LIN {X 0,Y 467.586,Z 97.863,A -85,B 0,C 180,E1 -7602.569,E2 -7602.569} C_VEL
LIN {X 0,Y 467.57,Z 97.863,A -85,B 0,C 180,E1 -7605.055,E2 -7605.055} C_VEL
LIN {X 0,Y 467.589,Z 97.863,A -85,B 0,C 180,E1 -7607.442,E2 -7607.442} C_VEL
LIN {X 0,Y 467.56,Z 97.864,A -85,B 0,C 180,E1 -7610.855,E2 -7610.855} C_VEL
LIN {X 0,Y 467.56,Z 97.866,A -85,B 0,C 180,E1 -7614.263,E2 -7614.263} C_VEL
LIN {X 0,Y 467.582,Z 97.866,A -85,B 0,C 180,E1 -7617.323,E2 -7617.323} C_VEL
LIN {X 0,Y 467.57,Z 97.868,A -85,B 0,C 180,E1 -7620.67,E2 -7620.67} C_VEL
LIN {X 0,Y 467.644,Z 97.873,A -85,B 0,C 180,E1 -7622.313,E2 -7622.313} C_VEL
LIN {X 0,Y 470.573,Z 111.961,A -85,B 0,C 180,E1 -7624.81,E2 -7624.81} C_VEL
LIN {X 0,Y 470.522,Z 117.185,A -85,B 0,C 180,E1 -7625.665,E2 -7625.665} C_VEL
LIN {X 0,Y 469.718,Z 134.843,A -85,B 0,C 180,E1 -7628.497,E2 -7628.497} C_VEL
LIN {X 0,Y 469.444,Z 141.034,A -85,B 0,C 180,E1 -7629.471,E2 -7629.471} C_VEL
LIN {X 0,Y 473.187,Z 162.958,A -85,B 0,C 180,E1 -7629.971,E2 -7629.971} C_VEL
LIN {X 0,Y 471.968,Z 279.138,A -85,B 0,C 180,E1 -7631.779,E2 -7631.779} C_VEL
LIN {X 0,Y 471.559,Z 293.745,A -85,B 0,C 180,E1 -7632.184,E2 -7632.184} C_VEL
LIN {X 0,Y 471.065,Z 307.853,A -85,B 0,C 180,E1 -7632.759,E2 -7632.759} C_VEL
LIN {X 0,Y 470.402,Z 321.628,A -85,B 0,C 180,E1 -7633.51,E2 -7633.51} C_VEL
LIN {X 0,Y 469.751,Z 334.084,A -85,B 0,C 180,E1 -7634.379,E2 -7634.379} C_VEL
LIN {X 0,Y 469.073,Z 345.474,A -85,B 0,C 180,E1 -7635.356,E2 -7635.356} C_VEL
LIN {X 0,Y 468.461,Z 356.923,A -85,B 0,C 180,E1 -7636.555,E2 -7636.555} C_VEL
LIN {X 0,Y 467.959,Z 367.131,A -85,B 0,C 180,E1 -7637.864,E2 -7637.864} C_VEL
LIN {X 0,Y 467.506,Z 375.588,A -85,B 0,C 180,E1 -7639.17,E2 -7639.17} C_VEL
LIN {X 0,Y 467.122,Z 383.662,A -85,B 0,C 180,E1 -7640.694,E2 -7640.694} C_VEL
LIN {X 0,Y 466.853,Z 390.164,A -85,B 0,C 180,E1 -7642.215,E2 -7642.215} C_VEL
LIN {X 0,Y 466.709,Z 395.086,A -85,B 0,C 180,E1 -7643.66,E2 -7643.66} C_VEL
LIN {X 0,Y 466.721,Z 398.205,A -85,B 0,C 180,E1 -7644.818,E2 -7644.818} C_VEL
LIN {X 0,Y 466.652,Z 401.65,A -85,B 0,C 180,E1 -7646.548,E2 -7646.548} C_VEL
LIN {X 0,Y 466.607,Z 403.692,A -85,B 0,C 180,E1 -7648.275,E2 -7648.275} C_VEL
LIN {X 0,Y 466.601,Z 404.382,A -85,B 0,C 180,E1 -7650.001,E2 -7650.001} C_VEL
LIN {X 0,Y 466.607,Z 403.73,A -85,B 0,C 180,E1 -7651.727,E2 -7651.727} C_VEL
LIN {X 0,Y 466.653,Z 401.724,A -85,B 0,C 180,E1 -7653.455,E2 -7653.455} C_VEL
LIN {X 0,Y 466.722,Z 398.32,A -85,B 0,C 180,E1 -7655.185,E2 -7655.185} C_VEL
LIN {X 0,Y 466.827,Z 393.417,A -85,B 0,C 180,E1 -7656.919,E2 -7656.919} C_VEL
LIN {X 0,Y 467.025,Z 386.875,A -85,B 0,C 180,E1 -7658.656,E2 -7658.656} C_VEL
LIN {X 0,Y 467.304,Z 379.614,A -85,B 0,C 180,E1 -7660.18,E2 -7660.18} C_VEL
LIN {X 0,Y 467.839,Z 370.65,A -85,B 0,C 180,E1 -7661.702,E2 -7661.702} C_VEL
LIN {X 0,Y 468.33,Z 361.254,A -85,B 0,C 180,E1 -7663.01,E2 -7663.01} C_VEL
LIN {X 0,Y 468.911,Z 350.867,A -85,B 0,C 180,E1 -7664.208,E2 -7664.208} C_VEL
LIN {X 0,Y 469.603,Z 339.433,A -85,B 0,C 180,E1 -7665.295,E2 -7665.295} C_VEL
LIN {X 0,Y 470.358,Z 326.789,A -85,B 0,C 180,E1 -7666.271,E2 -7666.271} C_VEL
LIN {X 0,Y 471.062,Z 313.567,A -85,B 0,C 180,E1 -7667.08,E2 -7667.08} C_VEL
LIN {X 0,Y 471.608,Z 300.6,A -85,B 0,C 180,E1 -7667.694,E2 -7667.694} C_VEL
LIN {X 0,Y 472.129,Z 287.209,A -85,B 0,C 180,E1 -7668.155,E2 -7668.155} C_VEL
LIN {X 0,Y 472.522,Z 272.513,A -85,B 0,C 180,E1 -7668.482,E2 -7668.482} C_VEL
LIN {X 0,Y 473.546,Z 161.959,A -85,B 0,C 180,E1 -7670.211,E2 -7670.211} C_VEL
LIN {X 0,Y 469.646,Z 140.816,A -85,B 0,C 180,E1 -7670.746,E2 -7670.746} C_VEL
LIN {X 0,Y 470.621,Z 122.114,A -85,B 0,C 180,E1 -7673.78,E2 -7673.78} C_VEL
LIN {X 0,Y 471.062,Z 113.762,A -85,B 0,C 180,E1 -7675.165,E2 -7675.165} C_VEL
LIN {X 0,Y 468.091,Z 99.917,A -85,B 0,C 180,E1 -7677.74,E2 -7677.74} C_VEL
LIN {X 0,Y 467.62,Z 97.864,A -85,B 0,C 180,E1 -7678.136,E2 -7678.136} C_VEL
LIN {X 0,Y 467.593,Z 97.869,A -85,B 0,C 180,E1 -7681.741,E2 -7681.741} C_VEL
LIN {X 0,Y 467.568,Z 97.868,A -85,B 0,C 180,E1 -7684.834,E2 -7684.834} C_VEL
LIN {X 0,Y 467.574,Z 97.866,A -85,B 0,C 180,E1 -7688.045,E2 -7688.045} C_VEL
LIN {X 0,Y 467.586,Z 97.861,A -85,B 0,C 180,E1 -7691.403,E2 -7691.403} C_VEL
LIN {X 0,Y 467.579,Z 97.864,A -85,B 0,C 180,E1 -7695.052,E2 -7695.052} C_VEL
LIN {X 0,Y 467.588,Z 97.866,A -85,B 0,C 180,E1 -7697.438,E2 -7697.438} C_VEL
LIN {X 0,Y 467.582,Z 97.866,A -85,B 0,C 180,E1 -7700.047,E2 -7700.047} C_VEL
LIN {X 0,Y 467.537,Z 97.868,A -85,B 0,C 180,E1 -7703.036,E2 -7703.036} C_VEL
LIN {X 0,Y 467.582,Z 97.862,A -85,B 0,C 180,E1 -7706.209,E2 -7706.209} C_VEL
LIN {X 0,Y 467.581,Z 97.865,A -85,B 0,C 180,E1 -7709.265,E2 -7709.265} C_VEL
LIN {X 0,Y 467.617,Z 97.855,A -85,B 0,C 180,E1 -7712.468,E2 -7712.468} C_VEL
LIN {X 0,Y 467.596,Z 97.864,A -85,B 0,C 180,E1 -7715.11,E2 -7715.11} C_VEL
LIN {X 0,Y 467.547,Z 97.867,A -85,B 0,C 180,E1 -7717.925,E2 -7717.925} C_VEL
LIN {X 0,Y 467.634,Z 97.856,A -85,B 0,C 180,E1 -7720.69,E2 -7720.69} C_VEL
LIN {X 0,Y 467.65,Z 97.852,A -85,B 0,C 180,E1 -7724.303,E2 -7724.303} C_VEL
LIN {X 0,Y 467.668,Z 97.85,A -85,B 0,C 180,E1 -7727.852,E2 -7727.852} C_VEL
LIN {X 0,Y 467.677,Z 97.85,A -85,B 0,C 180,E1 -7731.355,E2 -7731.355} C_VEL
LIN {X 0,Y 467.721,Z 97.846,A -85,B 0,C 180,E1 -7733.96,E2 -7733.96} C_VEL
LIN {X 0,Y 467.858,Z 97.824,A -85,B 0,C 180,E1 -7737.414,E2 -7737.414} C_VEL
LIN {X 0,Y 467.887,Z 97.83,A -85,B 0,C 180,E1 -7739.997,E2 -7739.997} C_VEL
LIN {X 0,Y 467.857,Z 97.83,A -85,B 0,C 180,E1 -7742.58,E2 -7742.58} C_VEL
LIN {X 0,Y 467.725,Z 97.848,A -85,B 0,C 180,E1 -7746.035,E2 -7746.035} C_VEL
LIN {X 0,Y 467.672,Z 97.849,A -85,B 0,C 180,E1 -7748.64,E2 -7748.64} C_VEL
LIN {X 0,Y 467.658,Z 97.854,A -85,B 0,C 180,E1 -7752.142,E2 -7752.142} C_VEL
LIN {X 0,Y 467.638,Z 97.859,A -85,B 0,C 180,E1 -7755.692,E2 -7755.692} C_VEL
LIN {X 0,Y 467.619,Z 97.863,A -85,B 0,C 180,E1 -7759.304,E2 -7759.304} C_VEL
LIN {X 0,Y 467.53,Z 97.87,A -85,B 0,C 180,E1 -7762.07,E2 -7762.07} C_VEL
LIN {X 0,Y 467.563,Z 97.869,A -85,B 0,C 180,E1 -7764.886,E2 -7764.886} C_VEL
LIN {X 0,Y 467.608,Z 97.86,A -85,B 0,C 180,E1 -7767.766,E2 -7767.766} C_VEL
LIN {X 0,Y 467.557,Z 97.867,A -85,B 0,C 180,E1 -7771.041,E2 -7771.041} C_VEL
LIN {X 0,Y 467.565,Z 97.861,A -85,B 0,C 180,E1 -7774.236,E2 -7774.236} C_VEL
LIN {X 0,Y 467.532,Z 97.867,A -85,B 0,C 180,E1 -7777.182,E2 -7777.182} C_VEL
LIN {X 0,Y 467.558,Z 97.871,A -85,B 0,C 180,E1 -7780.261,E2 -7780.261} C_VEL
LIN {X 0,Y 467.569,Z 97.87,A -85,B 0,C 180,E1 -7782.563,E2 -7782.563} C_VEL
LIN {X 0,Y 467.546,Z 97.869,A -85,B 0,C 180,E1 -7785.049,E2 -7785.049} C_VEL
LIN {X 0,Y 467.551,Z 97.876,A -85,B 0,C 180,E1 -7788.593,E2 -7788.593} C_VEL
LIN {X 0,Y 467.605,Z 97.972,A -85,B 0,C 180,E1 -7789.323,E2 -7789.323} C_VEL
LIN {X 0,Y 469.891,Z 108.948,A -85,B 0,C 180,E1 -7791.631,E2 -7791.631} C_VEL
LIN {X 0,Y 470.21,Z 112.722,A -85,B 0,C 180,E1 -7792.381,E2 -7792.381} C_VEL
LIN {X 0,Y 469.959,Z 117.614,A -85,B 0,C 180,E1 -7793.306,E2 -7793.306} C_VEL
LIN {X 0,Y 473.812,Z 134.774,A -85,B 0,C 180,E1 -7793.792,E2 -7793.792} C_VEL
LIN {X 0,Y 472.582,Z 254.497,A -85,B 0,C 180,E1 -7795.685,E2 -7795.685} C_VEL
LIN {X 0,Y 472.2,Z 268.433,A -85,B 0,C 180,E1 -7796.073,E2 -7796.073} C_VEL
LIN {X 0,Y 472.044,Z 273.44,A -85,B 0,C 180,E1 -7796.253,E2 -7796.253} C_VEL
LIN {X 0,Y 471.249,Z 279.065,A -85,B 0,C 180,E1 -7796.453,E2 -7796.453} C_VEL
LIN {X 0,Y 468.134,Z 288.113,A -85,B 0,C 180,E1 -7796.775,E2 -7796.775} C_VEL
LIN {X 0,Y 464.937,Z 296.921,A -85,B 0,C 180,E1 -7797.179,E2 -7797.179} C_VEL
LIN {X 0,Y 464.02,Z 302.093,A -85,B 0,C 180,E1 -7797.502,E2 -7797.502} C_VEL
LIN {X 0,Y 463.276,Z 314.306,A -85,B 0,C 180,E1 -7798.461,E2 -7798.461} C_VEL
LIN {X 0,Y 462.579,Z 325.397,A -85,B 0,C 180,E1 -7799.53,E2 -7799.53} C_VEL
LIN {X 0,Y 461.928,Z 334.916,A -85,B 0,C 180,E1 -7800.631,E2 -7800.631} C_VEL
LIN {X 0,Y 461.223,Z 345.386,A -85,B 0,C 180,E1 -7802.093,E2 -7802.093} C_VEL
LIN {X 0,Y 460.703,Z 353.598,A -85,B 0,C 180,E1 -7803.498,E2 -7803.498} C_VEL
LIN {X 0,Y 460.305,Z 360.469,A -85,B 0,C 180,E1 -7804.931,E2 -7804.931} C_VEL
LIN {X 0,Y 459.964,Z 366.865,A -85,B 0,C 180,E1 -7806.591,E2 -7806.591} C_VEL
LIN {X 0,Y 459.825,Z 371.123,A -85,B 0,C 180,E1 -7808.008,E2 -7808.008} C_VEL
LIN {X 0,Y 459.653,Z 374.363,A -85,B 0,C 180,E1 -7809.41,E2 -7809.41} C_VEL
LIN {X 0,Y 459.492,Z 377.295,A -85,B 0,C 180,E1 -7811.263,E2 -7811.263} C_VEL
LIN {X 0,Y 459.422,Z 378.727,A -85,B 0,C 180,E1 -7813.102,E2 -7813.102} C_VEL
LIN {X 0,Y 459.471,Z 378.693,A -85,B 0,C 180,E1 -7814.927,E2 -7814.927} C_VEL
LIN {X 0,Y 459.477,Z 377.245,A -85,B 0,C 180,E1 -7816.735,E2 -7816.735} C_VEL
LIN {X 0,Y 459.622,Z 374.385,A -85,B 0,C 180,E1 -7818.533,E2 -7818.533} C_VEL
LIN {X 0,Y 459.756,Z 370.073,A -85,B 0,C 180,E1 -7820.319,E2 -7820.319} C_VEL
LIN {X 0,Y 460.008,Z 364.185,A -85,B 0,C 180,E1 -7822.095,E2 -7822.095} C_VEL
LIN {X 0,Y 460.358,Z 358.02,A -85,B 0,C 180,E1 -7823.544,E2 -7823.544} C_VEL
LIN {X 0,Y 460.723,Z 350.622,A -85,B 0,C 180,E1 -7824.967,E2 -7824.967} C_VEL
LIN {X 0,Y 461.238,Z 342.319,A -85,B 0,C 180,E1 -7826.286,E2 -7826.286} C_VEL
LIN {X 0,Y 461.841,Z 332.355,A -85,B 0,C 180,E1 -7827.6,E2 -7827.6} C_VEL
LIN {X 0,Y 462.503,Z 321.273,A -85,B 0,C 180,E1 -7828.802,E2 -7828.802} C_VEL
LIN {X 0,Y 463.207,Z 308.875,A -85,B 0,C 180,E1 -7829.89,E2 -7829.89} C_VEL
LIN {X 0,Y 463.947,Z 296.668,A -85,B 0,C 180,E1 -7830.752,E2 -7830.752} C_VEL
LIN {X 0,Y 464.499,Z 284.153,A -85,B 0,C 180,E1 -7831.456,E2 -7831.456} C_VEL
LIN {X 0,Y 464.951,Z 270.061,A -85,B 0,C 180,E1 -7832.056,E2 -7832.056} C_VEL
LIN {X 0,Y 465.269,Z 256.375,A -85,B 0,C 180,E1 -7832.461,E2 -7832.461} C_VEL
LIN {X 0,Y 465.598,Z 234.551,A -85,B 0,C 180,E1 -7832.838,E2 -7832.838} C_VEL
LIN {X 0,Y 466.531,Z 135.668,A -85,B 0,C 180,E1 -7834.384,E2 -7834.384} C_VEL
LIN {X 0,Y 462.773,Z 117.498,A -85,B 0,C 180,E1 -7834.858,E2 -7834.858} C_VEL
LIN {X 0,Y 462.996,Z 110.908,A -85,B 0,C 180,E1 -7836.098,E2 -7836.098} C_VEL
LIN {X 0,Y 460.643,Z 98.732,A -85,B 0,C 180,E1 -7838.592,E2 -7838.592} C_VEL
LIN {X 0,Y 460.633,Z 98.735,A -85,B 0,C 180,E1 -7842.478,E2 -7842.478} C_VEL
LIN {X 0,Y 460.583,Z 98.737,A -85,B 0,C 180,E1 -7846.007,E2 -7846.007} C_VEL
LIN {X 0,Y 460.538,Z 98.74,A -85,B 0,C 180,E1 -7848.904,E2 -7848.904} C_VEL
LIN {X 0,Y 460.527,Z 98.749,A -85,B 0,C 180,E1 -7851.484,E2 -7851.484} C_VEL
LIN {X 0,Y 460.522,Z 98.741,A -85,B 0,C 180,E1 -7854.332,E2 -7854.332} C_VEL
LIN {X 0,Y 460.548,Z 98.745,A -85,B 0,C 180,E1 -7857.244,E2 -7857.244} C_VEL
LIN {X 0,Y 460.498,Z 98.744,A -85,B 0,C 180,E1 -7860.239,E2 -7860.239} C_VEL
LIN {X 0,Y 460.495,Z 98.749,A -85,B 0,C 180,E1 -7863.326,E2 -7863.326} C_VEL
LIN {X 0,Y 460.475,Z 98.747,A -85,B 0,C 180,E1 -7866.018,E2 -7866.018} C_VEL
LIN {X 0,Y 460.559,Z 98.744,A -85,B 0,C 180,E1 -7868.907,E2 -7868.907} C_VEL
LIN {X 0,Y 460.517,Z 98.743,A -85,B 0,C 180,E1 -7872.18,E2 -7872.18} C_VEL
LIN {X 0,Y 460.525,Z 98.742,A -85,B 0,C 180,E1 -7875.418,E2 -7875.418} C_VEL
LIN {X 0,Y 460.516,Z 98.746,A -85,B 0,C 180,E1 -7878.397,E2 -7878.397} C_VEL
LIN {X 0,Y 460.523,Z 98.742,A -85,B 0,C 180,E1 -7881.272,E2 -7881.272} C_VEL
LIN {X 0,Y 460.487,Z 98.752,A -85,B 0,C 180,E1 -7884.557,E2 -7884.557} C_VEL
LIN {X 0,Y 460.507,Z 98.744,A -85,B 0,C 180,E1 -7887.718,E2 -7887.718} C_VEL
LIN {X 0,Y 460.523,Z 98.743,A -85,B 0,C 180,E1 -7890.772,E2 -7890.772} C_VEL
LIN {X 0,Y 460.561,Z 98.739,A -85,B 0,C 180,E1 -7893.739,E2 -7893.739} C_VEL
LIN {X 0,Y 460.539,Z 98.741,A -85,B 0,C 180,E1 -7896.628,E2 -7896.628} C_VEL
LIN {X 0,Y 460.553,Z 98.739,A -85,B 0,C 180,E1 -7899.457,E2 -7899.457} C_VEL
LIN {X 0,Y 460.541,Z 98.742,A -85,B 0,C 180,E1 -7902.233,E2 -7902.233} C_VEL
LIN {X 0,Y 460.552,Z 98.737,A -85,B 0,C 180,E1 -7904.968,E2 -7904.968} C_VEL
LIN {X 0,Y 460.613,Z 98.737,A -85,B 0,C 180,E1 -7907.669,E2 -7907.669} C_VEL
LIN {X 0,Y 460.616,Z 98.732,A -85,B 0,C 180,E1 -7911.227,E2 -7911.227} C_VEL
LIN {X 0,Y 460.701,Z 98.722,A -85,B 0,C 180,E1 -7913.873,E2 -7913.873} C_VEL
LIN {X 0,Y 460.815,Z 98.712,A -85,B 0,C 180,E1 -7917.381,E2 -7917.381} C_VEL
LIN {X 0,Y 460.842,Z 98.702,A -85,B 0,C 180,E1 -7920.003,E2 -7920.003} C_VEL
LIN {X 0,Y 460.816,Z 98.705,A -85,B 0,C 180,E1 -7922.625,E2 -7922.625} C_VEL
LIN {X 0,Y 460.701,Z 98.719,A -85,B 0,C 180,E1 -7926.133,E2 -7926.133} C_VEL
LIN {X 0,Y 460.621,Z 98.733,A -85,B 0,C 180,E1 -7928.779,E2 -7928.779} C_VEL
LIN {X 0,Y 460.606,Z 98.732,A -85,B 0,C 180,E1 -7932.448,E2 -7932.448} C_VEL
LIN {X 0,Y 460.594,Z 98.732,A -85,B 0,C 180,E1 -7936,E2 -7936} C_VEL
LIN {X 0,Y 460.566,Z 98.742,A -85,B 0,C 180,E1 -7938.904,E2 -7938.904} C_VEL
LIN {X 0,Y 460.511,Z 98.743,A -85,B 0,C 180,E1 -7941.488,E2 -7941.488} C_VEL
LIN {X 0,Y 460.539,Z 98.743,A -85,B 0,C 180,E1 -7944.335,E2 -7944.335} C_VEL
LIN {X 0,Y 460.581,Z 98.734,A -85,B 0,C 180,E1 -7947.245,E2 -7947.245} C_VEL
LIN {X 0,Y 460.508,Z 98.748,A -85,B 0,C 180,E1 -7950.242,E2 -7950.242} C_VEL
LIN {X 0,Y 460.527,Z 98.74,A -85,B 0,C 180,E1 -7953.327,E2 -7953.327} C_VEL
LIN {X 0,Y 460.476,Z 98.75,A -85,B 0,C 180,E1 -7956.532,E2 -7956.532} C_VEL
LIN {X 0,Y 460.531,Z 98.745,A -85,B 0,C 180,E1 -7959.865,E2 -7959.865} C_VEL
LIN {X 0,Y 460.512,Z 98.742,A -85,B 0,C 180,E1 -7962.902,E2 -7962.902} C_VEL
LIN {X 0,Y 460.509,Z 98.749,A -85,B 0,C 180,E1 -7965.833,E2 -7965.833} C_VEL
LIN {X 0,Y 460.531,Z 98.74,A -85,B 0,C 180,E1 -7968.991,E2 -7968.991} C_VEL
LIN {X 0,Y 460.519,Z 98.744,A -85,B 0,C 180,E1 -7971.268,E2 -7971.268} C_VEL
LIN {X 0,Y 460.511,Z 98.742,A -85,B 0,C 180,E1 -7974.556,E2 -7974.556} C_VEL
LIN {X 0,Y 460.532,Z 98.747,A -85,B 0,C 180,E1 -7977.717,E2 -7977.717} C_VEL
LIN {X 0,Y 460.54,Z 98.745,A -85,B 0,C 180,E1 -7980.771,E2 -7980.771} C_VEL
LIN {X 0,Y 460.602,Z 98.879,A -85,B 0,C 180,E1 -7982.094,E2 -7982.094} C_VEL
LIN {X 0,Y 463.594,Z 113.017,A -85,B 0,C 180,E1 -7984.644,E2 -7984.644} C_VEL
LIN {X 0,Y 463.751,Z 116.506,A -85,B 0,C 180,E1 -7985.234,E2 -7985.234} C_VEL
LIN {X 0,Y 462.737,Z 136.103,A -85,B 0,C 180,E1 -7988.424,E2 -7988.424} C_VEL
LIN {X 0,Y 462.521,Z 140.69,A -85,B 0,C 180,E1 -7989.164,E2 -7989.164} C_VEL
LIN {X 0,Y 466.435,Z 163.215,A -85,B 0,C 180,E1 -7989.702,E2 -7989.702} C_VEL
LIN {X 0,Y 465.217,Z 277.906,A -85,B 0,C 180,E1 -7991.505,E2 -7991.505} C_VEL
LIN {X 0,Y 464.833,Z 292.168,A -85,B 0,C 180,E1 -7991.888,E2 -7991.888} C_VEL
LIN {X 0,Y 464.265,Z 306.329,A -85,B 0,C 180,E1 -7992.455,E2 -7992.455} C_VEL
LIN {X 0,Y 463.639,Z 319.818,A -85,B 0,C 180,E1 -7993.182,E2 -7993.182} C_VEL
LIN {X 0,Y 462.962,Z 332.163,A -85,B 0,C 180,E1 -7994.031,E2 -7994.031} C_VEL
LIN {X 0,Y 462.252,Z 343.859,A -85,B 0,C 180,E1 -7995.022,E2 -7995.022} C_VEL
LIN {X 0,Y 461.592,Z 354.572,A -85,B 0,C 180,E1 -7996.126,E2 -7996.126} C_VEL
LIN {X 0,Y 461.074,Z 365.262,A -85,B 0,C 180,E1 -7997.465,E2 -7997.465} C_VEL
LIN {X 0,Y 460.553,Z 373.956,A -85,B 0,C 180,E1 -7998.782,E2 -7998.782} C_VEL
LIN {X 0,Y 460.116,Z 382.352,A -85,B 0,C 180,E1 -8000.329,E2 -8000.329} C_VEL
LIN {X 0,Y 459.846,Z 388.194,A -85,B 0,C 180,E1 -8001.653,E2 -8001.653} C_VEL
LIN {X 0,Y 459.735,Z 393.005,A -85,B 0,C 180,E1 -8002.977,E2 -8002.977} C_VEL
LIN {X 0,Y 459.628,Z 397.974,A -85,B 0,C 180,E1 -8004.737,E2 -8004.737} C_VEL
LIN {X 0,Y 459.55,Z 401.431,A -85,B 0,C 180,E1 -8006.494,E2 -8006.494} C_VEL
LIN {X 0,Y 459.52,Z 403.485,A -85,B 0,C 180,E1 -8008.248,E2 -8008.248} C_VEL
LIN {X 0,Y 459.533,Z 404.186,A -85,B 0,C 180,E1 -8010.001,E2 -8010.001} C_VEL
LIN {X 0,Y 459.52,Z 403.544,A -85,B 0,C 180,E1 -8011.754,E2 -8011.754} C_VEL
LIN {X 0,Y 459.549,Z 401.551,A -85,B 0,C 180,E1 -8013.508,E2 -8013.508} C_VEL
LIN {X 0,Y 459.63,Z 398.16,A -85,B 0,C 180,E1 -8015.265,E2 -8015.265} C_VEL
LIN {X 0,Y 459.738,Z 393.275,A -85,B 0,C 180,E1 -8017.026,E2 -8017.026} C_VEL
LIN {X 0,Y 459.96,Z 386.758,A -85,B 0,C 180,E1 -8018.79,E2 -8018.79} C_VEL
LIN {X 0,Y 460.275,Z 379.516,A -85,B 0,C 180,E1 -8020.337,E2 -8020.337} C_VEL
LIN {X 0,Y 460.832,Z 370.578,A -85,B 0,C 180,E1 -8021.882,E2 -8021.882} C_VEL
LIN {X 0,Y 461.349,Z 361.212,A -85,B 0,C 180,E1 -8023.21,E2 -8023.21} C_VEL
LIN {X 0,Y 462.004,Z 350.859,A -85,B 0,C 180,E1 -8024.425,E2 -8024.425} C_VEL
LIN {X 0,Y 462.719,Z 339.465,A -85,B 0,C 180,E1 -8025.528,E2 -8025.528} C_VEL
LIN {X 0,Y 463.549,Z 326.897,A -85,B 0,C 180,E1 -8026.517,E2 -8026.517} C_VEL
LIN {X 0,Y 464.269,Z 314.085,A -85,B 0,C 180,E1 -8027.321,E2 -8027.321} C_VEL
LIN {X 0,Y 464.928,Z 300.065,A -85,B 0,C 180,E1 -8027.997,E2 -8027.997} C_VEL
LIN {X 0,Y 465.476,Z 285.848,A -85,B 0,C 180,E1 -8028.487,E2 -8028.487} C_VEL
LIN {X 0,Y 465.878,Z 272.232,A -85,B 0,C 180,E1 -8028.784,E2 -8028.784} C_VEL
LIN {X 0,Y 467.066,Z 163.619,A -85,B 0,C 180,E1 -8030.502,E2 -8030.502} C_VEL
LIN {X 0,Y 463.42,Z 143.666,A -85,B 0,C 180,E1 -8031.017,E2 -8031.017} C_VEL
LIN {X 0,Y 462.796,Z 140.399,A -85,B 0,C 180,E1 -8031.119,E2 -8031.119} C_VEL
LIN {X 0,Y 463.853,Z 122.146,A -85,B 0,C 180,E1 -8034.149,E2 -8034.149} C_VEL
LIN {X 0,Y 464.183,Z 115.204,A -85,B 0,C 180,E1 -8035.324,E2 -8035.324} C_VEL
LIN {X 0,Y 461.509,Z 102.63,A -85,B 0,C 180,E1 -8037.702,E2 -8037.702} C_VEL
LIN {X 0,Y 460.584,Z 98.739,A -85,B 0,C 180,E1 -8038.48,E2 -8038.48} C_VEL
LIN {X 0,Y 460.532,Z 98.748,A -85,B 0,C 180,E1 -8041.283,E2 -8041.283} C_VEL
LIN {X 0,Y 460.534,Z 98.744,A -85,B 0,C 180,E1 -8044.504,E2 -8044.504} C_VEL
LIN {X 0,Y 460.511,Z 98.743,A -85,B 0,C 180,E1 -8047.624,E2 -8047.624} C_VEL
LIN {X 0,Y 460.54,Z 98.738,A -85,B 0,C 180,E1 -8051.012,E2 -8051.012} C_VEL
LIN {X 0,Y 460.525,Z 98.743,A -85,B 0,C 180,E1 -8054.589,E2 -8054.589} C_VEL
LIN {X 0,Y 460.527,Z 98.738,A -85,B 0,C 180,E1 -8057.817,E2 -8057.817} C_VEL
LIN {X 0,Y 460.531,Z 98.743,A -85,B 0,C 180,E1 -8060.135,E2 -8060.135} C_VEL
LIN {X 0,Y 460.486,Z 98.75,A -85,B 0,C 180,E1 -8063.469,E2 -8063.469} C_VEL
LIN {X 0,Y 460.532,Z 98.74,A -85,B 0,C 180,E1 -8066.673,E2 -8066.673} C_VEL
LIN {X 0,Y 460.52,Z 98.745,A -85,B 0,C 180,E1 -8069.759,E2 -8069.759} C_VEL
LIN {X 0,Y 460.548,Z 98.738,A -85,B 0,C 180,E1 -8072.752,E2 -8072.752} C_VEL
LIN {X 0,Y 460.542,Z 98.736,A -85,B 0,C 180,E1 -8075.665,E2 -8075.665} C_VEL
LIN {X 0,Y 460.535,Z 98.744,A -85,B 0,C 180,E1 -8078.577,E2 -8078.577} C_VEL
LIN {X 0,Y 460.597,Z 98.736,A -85,B 0,C 180,E1 -8081.309,E2 -8081.309} C_VEL
LIN {X 0,Y 460.617,Z 98.727,A -85,B 0,C 180,E1 -8084.057,E2 -8084.057} C_VEL
LIN {X 0,Y 460.621,Z 98.727,A -85,B 0,C 180,E1 -8087.664,E2 -8087.664} C_VEL
LIN {X 0,Y 460.628,Z 98.728,A -85,B 0,C 180,E1 -8091.221,E2 -8091.221} C_VEL
LIN {X 0,Y 460.686,Z 98.721,A -85,B 0,C 180,E1 -8093.867,E2 -8093.867} C_VEL
LIN {X 0,Y 460.799,Z 98.703,A -85,B 0,C 180,E1 -8097.375,E2 -8097.375} C_VEL
LIN {X 0,Y 460.857,Z 98.706,A -85,B 0,C 180,E1 -8099.997,E2 -8099.997} C_VEL
LIN {X 0,Y 460.797,Z 98.709,A -85,B 0,C 180,E1 -8102.62,E2 -8102.62} C_VEL
LIN {X 0,Y 460.689,Z 98.725,A -85,B 0,C 180,E1 -8106.127,E2 -8106.127} C_VEL
LIN {X 0,Y 460.623,Z 98.727,A -85,B 0,C 180,E1 -8108.773,E2 -8108.773} C_VEL
LIN {X 0,Y 460.611,Z 98.73,A -85,B 0,C 180,E1 -8112.331,E2 -8112.331} C_VEL
LIN {X 0,Y 460.6,Z 98.732,A -85,B 0,C 180,E1 -8115.994,E2 -8115.994} C_VEL
LIN {X 0,Y 460.565,Z 98.738,A -85,B 0,C 180,E1 -8119.612,E2 -8119.612} C_VEL
LIN {X 0,Y 460.506,Z 98.744,A -85,B 0,C 180,E1 -8122.425,E2 -8122.425} C_VEL
LIN {X 0,Y 460.539,Z 98.739,A -85,B 0,C 180,E1 -8125.792,E2 -8125.792} C_VEL
LIN {X 0,Y 460.541,Z 98.74,A -85,B 0,C 180,E1 -8128.229,E2 -8128.229} C_VEL
LIN {X 0,Y 460.51,Z 98.748,A -85,B 0,C 180,E1 -8131.279,E2 -8131.279} C_VEL
LIN {X 0,Y 460.51,Z 98.74,A -85,B 0,C 180,E1 -8134.5,E2 -8134.5} C_VEL
LIN {X 0,Y 460.486,Z 98.743,A -85,B 0,C 180,E1 -8137.619,E2 -8137.619} C_VEL
LIN {X 0,Y 460.522,Z 98.747,A -85,B 0,C 180,E1 -8140.265,E2 -8140.265} C_VEL
LIN {X 0,Y 460.48,Z 98.75,A -85,B 0,C 180,E1 -8143.372,E2 -8143.372} C_VEL
LIN {X 0,Y 460.488,Z 98.754,A -85,B 0,C 180,E1 -8146.622,E2 -8146.622} C_VEL
LIN {X 0,Y 460.555,Z 98.89,A -85,B 0,C 180,E1 -8149.024,E2 -8149.024} C_VEL
LIN {X 0,Y 463.004,Z 110.519,A -85,B 0,C 180,E1 -8151.511,E2 -8151.511} C_VEL
LIN {X 0,Y 463.325,Z 114.669,A -85,B 0,C 180,E1 -8152.348,E2 -8152.348} C_VEL
LIN {X 0,Y 463.133,Z 117.901,A -85,B 0,C 180,E1 -8152.967,E2 -8152.967} C_VEL
LIN {X 0,Y 467.31,Z 136.33,A -85,B 0,C 180,E1 -8153.49,E2 -8153.49} C_VEL
LIN {X 0,Y 465.932,Z 254.799,A -85,B 0,C 180,E1 -8155.388,E2 -8155.388} C_VEL
LIN {X 0,Y 465.545,Z 268.701,A -85,B 0,C 180,E1 -8155.781,E2 -8155.781} C_VEL
LIN {X 0,Y 465.038,Z 282.141,A -85,B 0,C 180,E1 -8156.333,E2 -8156.333} C_VEL
LIN {X 0,Y 464.336,Z 296.242,A -85,B 0,C 180,E1 -8157.111,E2 -8157.111} C_VEL
LIN {X 0,Y 464.02,Z 302.093,A -85,B 0,C 180,E1 -8157.502,E2 -8157.502} C_VEL
LIN {X 0,Y 463.111,Z 307.223,A -85,B 0,C 180,E1 -8157.852,E2 -8157.852} C_VEL
LIN {X 0,Y 459.89,Z 315.403,A -85,B 0,C 180,E1 -8158.417,E2 -8158.417} C_VEL
LIN {X 0,Y 456.59,Z 323.242,A -85,B 0,C 180,E1 -8159.055,E2 -8159.055} C_VEL
LIN {X 0,Y 455.571,Z 327.76,A -85,B 0,C 180,E1 -8159.513,E2 -8159.513} C_VEL
LIN {X 0,Y 454.929,Z 336.909,A -85,B 0,C 180,E1 -8160.626,E2 -8160.626} C_VEL
LIN {X 0,Y 454.193,Z 346.884,A -85,B 0,C 180,E1 -8162.093,E2 -8162.093} C_VEL
LIN {X 0,Y 453.587,Z 355.724,A -85,B 0,C 180,E1 -8163.697,E2 -8163.697} C_VEL
LIN {X 0,Y 453.139,Z 362.605,A -85,B 0,C 180,E1 -8165.243,E2 -8165.243} C_VEL
LIN {X 0,Y 452.89,Z 367.88,A -85,B 0,C 180,E1 -8166.713,E2 -8166.713} C_VEL
LIN {X 0,Y 452.736,Z 371.923,A -85,B 0,C 180,E1 -8168.125,E2 -8168.125} C_VEL
LIN {X 0,Y 452.607,Z 374.082,A -85,B 0,C 180,E1 -8169.074,E2 -8169.074} C_VEL
LIN {X 0,Y 452.402,Z 377.194,A -85,B 0,C 180,E1 -8170.959,E2 -8170.959} C_VEL
LIN {X 0,Y 452.327,Z 378.799,A -85,B 0,C 180,E1 -8172.829,E2 -8172.829} C_VEL
LIN {X 0,Y 452.383,Z 378.963,A -85,B 0,C 180,E1 -8174.685,E2 -8174.685} C_VEL
LIN {X 0,Y 452.376,Z 377.721,A -85,B 0,C 180,E1 -8176.523,E2 -8176.523} C_VEL
LIN {X 0,Y 452.528,Z 375.04,A -85,B 0,C 180,E1 -8178.351,E2 -8178.351} C_VEL
LIN {X 0,Y 452.655,Z 370.903,A -85,B 0,C 180,E1 -8180.165,E2 -8180.165} C_VEL
LIN {X 0,Y 452.907,Z 365.201,A -85,B 0,C 180,E1 -8181.971,E2 -8181.971} C_VEL
LIN {X 0,Y 453.278,Z 359.02,A -85,B 0,C 180,E1 -8183.49,E2 -8183.49} C_VEL
LIN {X 0,Y 453.699,Z 350.836,A -85,B 0,C 180,E1 -8185.111,E2 -8185.111} C_VEL
LIN {X 0,Y 454.267,Z 342.53,A -85,B 0,C 180,E1 -8186.451,E2 -8186.451} C_VEL
LIN {X 0,Y 454.893,Z 332.564,A -85,B 0,C 180,E1 -8187.785,E2 -8187.785} C_VEL
LIN {X 0,Y 455.586,Z 321.471,A -85,B 0,C 180,E1 -8189.004,E2 -8189.004} C_VEL
LIN {X 0,Y 456.332,Z 308.914,A -85,B 0,C 180,E1 -8190.12,E2 -8190.12} C_VEL
LIN {X 0,Y 457.12,Z 295.753,A -85,B 0,C 180,E1 -8191.052,E2 -8191.052} C_VEL
LIN {X 0,Y 457.736,Z 283.043,A -85,B 0,C 180,E1 -8191.758,E2 -8191.758} C_VEL
LIN {X 0,Y 458.179,Z 268.659,A -85,B 0,C 180,E1 -8192.361,E2 -8192.361} C_VEL
LIN {X 0,Y 458.549,Z 254.092,A -85,B 0,C 180,E1 -8192.771,E2 -8192.771} C_VEL
LIN {X 0,Y 459.848,Z 136.88,A -85,B 0,C 180,E1 -8194.647,E2 -8194.647} C_VEL
LIN {X 0,Y 455.871,Z 117.738,A -85,B 0,C 180,E1 -8195.144,E2 -8195.144} C_VEL
LIN {X 0,Y 456.072,Z 112.259,A -85,B 0,C 180,E1 -8196.191,E2 -8196.191} C_VEL
LIN {X 0,Y 453.582,Z 99.611,A -85,B 0,C 180,E1 -8198.82,E2 -8198.82} C_VEL
LIN {X 0,Y 453.602,Z 99.611,A -85,B 0,C 180,E1 -8202.572,E2 -8202.572} C_VEL
LIN {X 0,Y 453.52,Z 99.615,A -85,B 0,C 180,E1 -8206.195,E2 -8206.195} C_VEL
LIN {X 0,Y 453.487,Z 99.619,A -85,B 0,C 180,E1 -8209.043,E2 -8209.043} C_VEL
LIN {X 0,Y 453.468,Z 99.623,A -85,B 0,C 180,E1 -8211.835,E2 -8211.835} C_VEL
LIN {X 0,Y 453.496,Z 99.617,A -85,B 0,C 180,E1 -8214.734,E2 -8214.734} C_VEL
LIN {X 0,Y 453.502,Z 99.616,A -85,B 0,C 180,E1 -8217.962,E2 -8217.962} C_VEL
LIN {X 0,Y 453.45,Z 99.625,A -85,B 0,C 180,E1 -8220.76,E2 -8220.76} C_VEL
LIN {X 0,Y 453.446,Z 99.623,A -85,B 0,C 180,E1 -8223.914,E2 -8223.914} C_VEL
LIN {X 0,Y 453.447,Z 99.628,A -85,B 0,C 180,E1 -8227.188,E2 -8227.188} C_VEL
LIN {X 0,Y 453.511,Z 99.616,A -85,B 0,C 180,E1 -8229.446,E2 -8229.446} C_VEL
LIN {X 0,Y 453.468,Z 99.625,A -85,B 0,C 180,E1 -8232.992,E2 -8232.992} C_VEL
LIN {X 0,Y 453.511,Z 99.614,A -85,B 0,C 180,E1 -8235.791,E2 -8235.791} C_VEL
LIN {X 0,Y 453.487,Z 99.618,A -85,B 0,C 180,E1 -8239.408,E2 -8239.408} C_VEL
LIN {X 0,Y 453.451,Z 99.626,A -85,B 0,C 180,E1 -8242.224,E2 -8242.224} C_VEL
LIN {X 0,Y 453.462,Z 99.621,A -85,B 0,C 180,E1 -8245.225,E2 -8245.225} C_VEL
LIN {X 0,Y 453.459,Z 99.627,A -85,B 0,C 180,E1 -8248.473,E2 -8248.473} C_VEL
LIN {X 0,Y 453.491,Z 99.617,A -85,B 0,C 180,E1 -8251.291,E2 -8251.291} C_VEL
LIN {X 0,Y 453.532,Z 99.618,A -85,B 0,C 180,E1 -8254.289,E2 -8254.289} C_VEL
LIN {X 0,Y 453.48,Z 99.618,A -85,B 0,C 180,E1 -8257.208,E2 -8257.208} C_VEL
LIN {X 0,Y 453.508,Z 99.621,A -85,B 0,C 180,E1 -8260.07,E2 -8260.07} C_VEL
LIN {X 0,Y 453.491,Z 99.617,A -85,B 0,C 180,E1 -8262.879,E2 -8262.879} C_VEL
LIN {X 0,Y 453.498,Z 99.622,A -85,B 0,C 180,E1 -8265.647,E2 -8265.647} C_VEL
LIN {X 0,Y 453.564,Z 99.609,A -85,B 0,C 180,E1 -8268.382,E2 -8268.382} C_VEL
LIN {X 0,Y 453.637,Z 99.602,A -85,B 0,C 180,E1 -8271.988,E2 -8271.988} C_VEL
LIN {X 0,Y 453.663,Z 99.596,A -85,B 0,C 180,E1 -8274.67,E2 -8274.67} C_VEL
LIN {X 0,Y 453.756,Z 99.591,A -85,B 0,C 180,E1 -8277.34,E2 -8277.34} C_VEL
LIN {X 0,Y 453.813,Z 99.578,A -85,B 0,C 180,E1 -8280.003,E2 -8280.003} C_VEL
LIN {X 0,Y 453.756,Z 99.585,A -85,B 0,C 180,E1 -8282.666,E2 -8282.666} C_VEL
LIN {X 0,Y 453.669,Z 99.595,A -85,B 0,C 180,E1 -8286.228,E2 -8286.228} C_VEL
LIN {X 0,Y 453.584,Z 99.611,A -85,B 0,C 180,E1 -8288.916,E2 -8288.916} C_VEL
LIN {X 0,Y 453.556,Z 99.611,A -85,B 0,C 180,E1 -8292.532,E2 -8292.532} C_VEL
LIN {X 0,Y 453.539,Z 99.612,A -85,B 0,C 180,E1 -8296.199,E2 -8296.199} C_VEL
LIN {X 0,Y 453.515,Z 99.618,A -85,B 0,C 180,E1 -8299.043,E2 -8299.043} C_VEL
LIN {X 0,Y 453.472,Z 99.619,A -85,B 0,C 180,E1 -8301.839,E2 -8301.839} C_VEL
LIN {X 0,Y 453.511,Z 99.62,A -85,B 0,C 180,E1 -8304.737,E2 -8304.737} C_VEL
LIN {X 0,Y 453.534,Z 99.613,A -85,B 0,C 180,E1 -8307.963,E2 -8307.963} C_VEL
LIN {X 0,Y 453.463,Z 99.621,A -85,B 0,C 180,E1 -8311.527,E2 -8311.527} C_VEL
LIN {X 0,Y 453.487,Z 99.619,A -85,B 0,C 180,E1 -8314.78,E2 -8314.78} C_VEL
LIN {X 0,Y 453.463,Z 99.626,A -85,B 0,C 180,E1 -8318.314,E2 -8318.314} C_VEL
LIN {X 0,Y 453.493,Z 99.618,A -85,B 0,C 180,E1 -8320.611,E2 -8320.611} C_VEL
LIN {X 0,Y 453.455,Z 99.622,A -85,B 0,C 180,E1 -8323.246,E2 -8323.246} C_VEL
LIN {X 0,Y 453.464,Z 99.626,A -85,B 0,C 180,E1 -8325.781,E2 -8325.781} C_VEL
LIN {X 0,Y 453.479,Z 99.622,A -85,B 0,C 180,E1 -8328.211,E2 -8328.211} C_VEL
LIN {X 0,Y 453.472,Z 99.619,A -85,B 0,C 180,E1 -8330.799,E2 -8330.799} C_VEL
LIN {X 0,Y 453.455,Z 99.626,A -85,B 0,C 180,E1 -8333.919,E2 -8333.919} C_VEL
LIN {X 0,Y 453.483,Z 99.621,A -85,B 0,C 180,E1 -8337.153,E2 -8337.153} C_VEL
LIN {X 0,Y 453.475,Z 99.624,A -85,B 0,C 180,E1 -8340.27,E2 -8340.27} C_VEL
LIN {X 0,Y 453.538,Z 99.695,A -85,B 0,C 180,E1 -8341.84,E2 -8341.84} C_VEL
LIN {X 0,Y 456.58,Z 114.037,A -85,B 0,C 180,E1 -8344.471,E2 -8344.471} C_VEL
LIN {X 0,Y 456.927,Z 116.578,A -85,B 0,C 180,E1 -8344.918,E2 -8344.918} C_VEL
LIN {X 0,Y 455.777,Z 136.95,A -85,B 0,C 180,E1 -8348.281,E2 -8348.281} C_VEL
LIN {X 0,Y 455.6,Z 140.516,A -85,B 0,C 180,E1 -8348.866,E2 -8348.866} C_VEL
LIN {X 0,Y 459.708,Z 164.556,A -85,B 0,C 180,E1 -8349.445,E2 -8349.445} C_VEL
LIN {X 0,Y 458.396,Z 278.976,A -85,B 0,C 180,E1 -8351.278,E2 -8351.278} C_VEL
LIN {X 0,Y 457.952,Z 293.523,A -85,B 0,C 180,E1 -8351.693,E2 -8351.693} C_VEL
LIN {X 0,Y 457.385,Z 307.133,A -85,B 0,C 180,E1 -8352.26,E2 -8352.26} C_VEL
LIN {X 0,Y 456.739,Z 320.478,A -85,B 0,C 180,E1 -8353.002,E2 -8353.002} C_VEL
LIN {X 0,Y 455.977,Z 333.093,A -85,B 0,C 180,E1 -8353.894,E2 -8353.894} C_VEL
LIN {X 0,Y 455.171,Z 345.788,A -85,B 0,C 180,E1 -8355.013,E2 -8355.013} C_VEL
LIN {X 0,Y 454.517,Z 356.145,A -85,B 0,C 180,E1 -8356.134,E2 -8356.134} C_VEL
LIN {X 0,Y 453.976,Z 366.439,A -85,B 0,C 180,E1 -8357.484,E2 -8357.484} C_VEL
LIN {X 0,Y 453.445,Z 374.956,A -85,B 0,C 180,E1 -8358.83,E2 -8358.83} C_VEL
LIN {X 0,Y 453.032,Z 383.084,A -85,B 0,C 180,E1 -8360.401,E2 -8360.401} C_VEL
LIN {X 0,Y 452.721,Z 389.629,A -85,B 0,C 180,E1 -8361.97,E2 -8361.97} C_VEL
LIN {X 0,Y 452.583,Z 394.17,A -85,B 0,C 180,E1 -8363.314,E2 -8363.314} C_VEL
LIN {X 0,Y 452.537,Z 397.726,A -85,B 0,C 180,E1 -8364.655,E2 -8364.655} C_VEL
LIN {X 0,Y 452.448,Z 401.2,A -85,B 0,C 180,E1 -8366.439,E2 -8366.439} C_VEL
LIN {X 0,Y 452.502,Z 402.409,A -85,B 0,C 180,E1 -8367.331,E2 -8367.331} C_VEL
LIN {X 0,Y 452.428,Z 403.796,A -85,B 0,C 180,E1 -8369.111,E2 -8369.111} C_VEL
LIN {X 0,Y 452.428,Z 403.842,A -85,B 0,C 180,E1 -8370.891,E2 -8370.891} C_VEL
LIN {X 0,Y 452.503,Z 402.548,A -85,B 0,C 180,E1 -8372.672,E2 -8372.672} C_VEL
LIN {X 0,Y 452.471,Z 399.879,A -85,B 0,C 180,E1 -8374.455,E2 -8374.455} C_VEL
LIN {X 0,Y 452.57,Z 395.771,A -85,B 0,C 180,E1 -8376.242,E2 -8376.242} C_VEL
LIN {X 0,Y 452.744,Z 390.106,A -85,B 0,C 180,E1 -8378.032,E2 -8378.032} C_VEL
LIN {X 0,Y 453.055,Z 383.729,A -85,B 0,C 180,E1 -8379.601,E2 -8379.601} C_VEL
LIN {X 0,Y 453.514,Z 375.81,A -85,B 0,C 180,E1 -8381.171,E2 -8381.171} C_VEL
LIN {X 0,Y 454.048,Z 366.797,A -85,B 0,C 180,E1 -8382.633,E2 -8382.633} C_VEL
LIN {X 0,Y 454.636,Z 357.639,A -85,B 0,C 180,E1 -8383.865,E2 -8383.865} C_VEL
LIN {X 0,Y 455.386,Z 346.632,A -85,B 0,C 180,E1 -8385.097,E2 -8385.097} C_VEL
LIN {X 0,Y 456.297,Z 334.387,A -85,B 0,C 180,E1 -8386.212,E2 -8386.212} C_VEL
LIN {X 0,Y 457.089,Z 321.518,A -85,B 0,C 180,E1 -8387.152,E2 -8387.152} C_VEL
LIN {X 0,Y 457.872,Z 307.747,A -85,B 0,C 180,E1 -8387.937,E2 -8387.937} C_VEL
LIN {X 0,Y 458.49,Z 293.396,A -85,B 0,C 180,E1 -8388.547,E2 -8388.547} C_VEL
LIN {X 0,Y 459.039,Z 279.106,A -85,B 0,C 180,E1 -8388.959,E2 -8388.959} C_VEL
LIN {X 0,Y 459.859,Z 218.509,A -85,B 0,C 180,E1 -8389.953,E2 -8389.953} C_VEL
LIN {X 0,Y 460.4,Z 163.646,A -85,B 0,C 180,E1 -8390.84,E2 -8390.84} C_VEL
LIN {X 0,Y 456.742,Z 144.122,A -85,B 0,C 180,E1 -8391.364,E2 -8391.364} C_VEL
LIN {X 0,Y 455.964,Z 140.166,A -85,B 0,C 180,E1 -8391.492,E2 -8391.492} C_VEL
LIN {X 0,Y 457.111,Z 122.198,A -85,B 0,C 180,E1 -8394.528,E2 -8394.528} C_VEL
LIN {X 0,Y 457.308,Z 116.642,A -85,B 0,C 180,E1 -8395.488,E2 -8395.488} C_VEL
LIN {X 0,Y 454.965,Z 105.629,A -85,B 0,C 180,E1 -8397.609,E2 -8397.609} C_VEL
LIN {X 0,Y 453.518,Z 99.618,A -85,B 0,C 180,E1 -8398.839,E2 -8398.839} C_VEL
LIN {X 0,Y 453.475,Z 99.628,A -85,B 0,C 180,E1 -8401.8,E2 -8401.8} C_VEL
LIN {X 0,Y 453.488,Z 99.622,A -85,B 0,C 180,E1 -8404.99,E2 -8404.99} C_VEL
LIN {X 0,Y 453.47,Z 99.626,A -85,B 0,C 180,E1 -8408.312,E2 -8408.312} C_VEL
LIN {X 0,Y 453.507,Z 99.614,A -85,B 0,C 180,E1 -8410.609,E2 -8410.609} C_VEL
LIN {X 0,Y 453.473,Z 99.625,A -85,B 0,C 180,E1 -8414.222,E2 -8414.222} C_VEL
LIN {X 0,Y 453.475,Z 99.622,A -85,B 0,C 180,E1 -8417.004,E2 -8417.004} C_VEL
LIN {X 0,Y 453.507,Z 99.608,A -85,B 0,C 180,E1 -8419.409,E2 -8419.409} C_VEL
LIN {X 0,Y 453.463,Z 99.62,A -85,B 0,C 180,E1 -8422.809,E2 -8422.809} C_VEL
LIN {X 0,Y 453.481,Z 99.619,A -85,B 0,C 180,E1 -8426.086,E2 -8426.086} C_VEL
LIN {X 0,Y 453.489,Z 99.62,A -85,B 0,C 180,E1 -8429.239,E2 -8429.239} C_VEL
LIN {X 0,Y 453.521,Z 99.611,A -85,B 0,C 180,E1 -8432.294,E2 -8432.294} C_VEL
LIN {X 0,Y 453.513,Z 99.616,A -85,B 0,C 180,E1 -8435.263,E2 -8435.263} C_VEL
LIN {X 0,Y 453.494,Z 99.619,A -85,B 0,C 180,E1 -8438.413,E2 -8438.413} C_VEL
LIN {X 0,Y 453.535,Z 99.617,A -85,B 0,C 180,E1 -8441.007,E2 -8441.007} C_VEL
LIN {X 0,Y 453.582,Z 99.602,A -85,B 0,C 180,E1 -8443.878,E2 -8443.878} C_VEL
LIN {X 0,Y 453.576,Z 99.605,A -85,B 0,C 180,E1 -8447.469,E2 -8447.469} C_VEL
LIN {X 0,Y 453.594,Z 99.605,A -85,B 0,C 180,E1 -8451.084,E2 -8451.084} C_VEL
LIN {X 0,Y 453.652,Z 99.597,A -85,B 0,C 180,E1 -8453.772,E2 -8453.772} C_VEL
LIN {X 0,Y 453.743,Z 99.582,A -85,B 0,C 180,E1 -8457.334,E2 -8457.334} C_VEL
LIN {X 0,Y 453.827,Z 99.581,A -85,B 0,C 180,E1 -8459.997,E2 -8459.997} C_VEL
LIN {X 0,Y 453.741,Z 99.588,A -85,B 0,C 180,E1 -8462.66,E2 -8462.66} C_VEL
LIN {X 0,Y 453.655,Z 99.601,A -85,B 0,C 180,E1 -8466.222,E2 -8466.222} C_VEL
LIN {X 0,Y 453.588,Z 99.604,A -85,B 0,C 180,E1 -8468.91,E2 -8468.91} C_VEL
LIN {X 0,Y 453.566,Z 99.607,A -85,B 0,C 180,E1 -8472.525,E2 -8472.525} C_VEL
LIN {X 0,Y 453.544,Z 99.609,A -85,B 0,C 180,E1 -8476.192,E2 -8476.192} C_VEL
LIN {X 0,Y 453.514,Z 99.619,A -85,B 0,C 180,E1 -8479.035,E2 -8479.035} C_VEL
LIN {X 0,Y 453.473,Z 99.622,A -85,B 0,C 180,E1 -8481.832,E2 -8481.832} C_VEL
LIN {X 0,Y 453.486,Z 99.621,A -85,B 0,C 180,E1 -8484.732,E2 -8484.732} C_VEL
LIN {X 0,Y 453.521,Z 99.615,A -85,B 0,C 180,E1 -8487.955,E2 -8487.955} C_VEL
LIN {X 0,Y 453.454,Z 99.625,A -85,B 0,C 180,E1 -8491.521,E2 -8491.521} C_VEL
LIN {X 0,Y 453.47,Z 99.619,A -85,B 0,C 180,E1 -8494.772,E2 -8494.772} C_VEL
LIN {X 0,Y 453.447,Z 99.622,A -85,B 0,C 180,E1 -8498.308,E2 -8498.308} C_VEL
LIN {X 0,Y 453.478,Z 99.621,A -85,B 0,C 180,E1 -8500.605,E2 -8500.605} C_VEL
LIN {X 0,Y 453.437,Z 99.628,A -85,B 0,C 180,E1 -8503.24,E2 -8503.24} C_VEL
LIN {X 0,Y 453.44,Z 99.626,A -85,B 0,C 180,E1 -8505.774,E2 -8505.774} C_VEL
LIN {X 0,Y 453.518,Z 99.798,A -85,B 0,C 180,E1 -8508.706,E2 -8508.706} C_VEL
LIN {X 0,Y 456.061,Z 111.805,A -85,B 0,C 180,E1 -8511.329,E2 -8511.329} C_VEL
LIN {X 0,Y 456.514,Z 114.962,A -85,B 0,C 180,E1 -8511.989,E2 -8511.989} C_VEL
LIN {X 0,Y 456.389,Z 118.299,A -85,B 0,C 180,E1 -8512.606,E2 -8512.606} C_VEL
LIN {X 0,Y 460.753,Z 137.386,A -85,B 0,C 180,E1 -8513.166,E2 -8513.166} C_VEL
LIN {X 0,Y 459.299,Z 255.112,A -85,B 0,C 180,E1 -8515.083,E2 -8515.083} C_VEL
LIN {X 0,Y 458.86,Z 269.379,A -85,B 0,C 180,E1 -8515.495,E2 -8515.495} C_VEL
LIN {X 0,Y 458.342,Z 282.597,A -85,B 0,C 180,E1 -8516.05,E2 -8516.05} C_VEL
LIN {X 0,Y 457.614,Z 296.474,A -85,B 0,C 180,E1 -8516.829,E2 -8516.829} C_VEL
LIN {X 0,Y 456.819,Z 309.72,A -85,B 0,C 180,E1 -8517.787,E2 -8517.787} C_VEL
LIN {X 0,Y 455.985,Z 322.125,A -85,B 0,C 180,E1 -8518.912,E2 -8518.912} C_VEL
LIN {X 0,Y 455.571,Z 327.76,A -85,B 0,C 180,E1 -8519.513,E2 -8519.513} C_VEL
LIN {X 0,Y 454.55,Z 332.181,A -85,B 0,C 180,E1 -8519.998,E2 -8519.998} C_VEL
LIN {X 0,Y 451.222,Z 339.102,A -85,B 0,C 180,E1 -8520.794,E2 -8520.794} C_VEL
LIN {X 0,Y 447.975,Z 345.598,A -85,B 0,C 180,E1 -8521.655,E2 -8521.655} C_VEL
LIN {X 0,Y 447.084,Z 349.201,A -85,B 0,C 180,E1 -8522.235,E2 -8522.235} C_VEL
LIN {X 0,Y 446.483,Z 357.588,A -85,B 0,C 180,E1 -8523.847,E2 -8523.847} C_VEL
LIN {X 0,Y 446.056,Z 363.772,A -85,B 0,C 180,E1 -8525.32,E2 -8525.32} C_VEL
LIN {X 0,Y 445.819,Z 368.757,A -85,B 0,C 180,E1 -8526.789,E2 -8526.789} C_VEL
LIN {X 0,Y 445.605,Z 373.282,A -85,B 0,C 180,E1 -8528.505,E2 -8528.505} C_VEL
LIN {X 0,Y 445.42,Z 375.647,A -85,B 0,C 180,E1 -8529.687,E2 -8529.687} C_VEL
LIN {X 0,Y 445.31,Z 378.167,A -85,B 0,C 180,E1 -8531.599,E2 -8531.599} C_VEL
LIN {X 0,Y 445.239,Z 379.215,A -85,B 0,C 180,E1 -8533.492,E2 -8533.492} C_VEL
LIN {X 0,Y 445.271,Z 378.839,A -85,B 0,C 180,E1 -8535.371,E2 -8535.371} C_VEL
LIN {X 0,Y 445.323,Z 377.066,A -85,B 0,C 180,E1 -8537.234,E2 -8537.234} C_VEL
LIN {X 0,Y 445.498,Z 373.877,A -85,B 0,C 180,E1 -8539.086,E2 -8539.086} C_VEL
LIN {X 0,Y 445.661,Z 369.173,A -85,B 0,C 180,E1 -8540.925,E2 -8540.925} C_VEL
LIN {X 0,Y 445.907,Z 364.585,A -85,B 0,C 180,E1 -8542.3,E2 -8542.3} C_VEL
LIN {X 0,Y 446.237,Z 357.97,A -85,B 0,C 180,E1 -8543.896,E2 -8543.896} C_VEL
LIN {X 0,Y 446.729,Z 349.759,A -85,B 0,C 180,E1 -8545.487,E2 -8545.487} C_VEL
LIN {X 0,Y 447.356,Z 341.187,A -85,B 0,C 180,E1 -8546.847,E2 -8546.847} C_VEL
LIN {X 0,Y 448.067,Z 330.836,A -85,B 0,C 180,E1 -8548.201,E2 -8548.201} C_VEL
LIN {X 0,Y 448.754,Z 320.455,A -85,B 0,C 180,E1 -8549.326,E2 -8549.326} C_VEL
LIN {X 0,Y 449.455,Z 309.184,A -85,B 0,C 180,E1 -8550.335,E2 -8550.335} C_VEL
LIN {X 0,Y 450.28,Z 296.019,A -85,B 0,C 180,E1 -8551.282,E2 -8551.282} C_VEL
LIN {X 0,Y 450.909,Z 283.15,A -85,B 0,C 180,E1 -8552.008,E2 -8552.008} C_VEL
LIN {X 0,Y 451.348,Z 269.488,A -85,B 0,C 180,E1 -8552.592,E2 -8552.592} C_VEL
LIN {X 0,Y 451.692,Z 255.322,A -85,B 0,C 180,E1 -8553.009,E2 -8553.009} C_VEL
LIN {X 0,Y 452.838,Z 164.005,A -85,B 0,C 180,E1 -8554.5,E2 -8554.5} C_VEL
LIN {X 0,Y 453.072,Z 137.708,A -85,B 0,C 180,E1 -8554.926,E2 -8554.926} C_VEL
LIN {X 0,Y 448.941,Z 117.946,A -85,B 0,C 180,E1 -8555.445,E2 -8555.445} C_VEL
LIN {X 0,Y 449.138,Z 113.586,A -85,B 0,C 180,E1 -8556.287,E2 -8556.287} C_VEL
LIN {X 0,Y 446.555,Z 100.486,A -85,B 0,C 180,E1 -8559.054,E2 -8559.054} C_VEL
LIN {X 0,Y 446.564,Z 100.488,A -85,B 0,C 180,E1 -8562.727,E2 -8562.727} C_VEL
LIN {X 0,Y 446.481,Z 100.492,A -85,B 0,C 180,E1 -8566.238,E2 -8566.238} C_VEL
LIN {X 0,Y 446.434,Z 100.501,A -85,B 0,C 180,E1 -8569.303,E2 -8569.303} C_VEL
LIN {X 0,Y 446.407,Z 100.5,A -85,B 0,C 180,E1 -8572.199,E2 -8572.199} C_VEL
LIN {X 0,Y 446.439,Z 100.5,A -85,B 0,C 180,E1 -8575.152,E2 -8575.152} C_VEL
LIN {X 0,Y 446.447,Z 100.494,A -85,B 0,C 180,E1 -8578.18,E2 -8578.18} C_VEL
LIN {X 0,Y 446.401,Z 100.506,A -85,B 0,C 180,E1 -8581.3,E2 -8581.3} C_VEL
LIN {X 0,Y 446.408,Z 100.501,A -85,B 0,C 180,E1 -8584.523,E2 -8584.523} C_VEL
LIN {X 0,Y 446.415,Z 100.498,A -85,B 0,C 180,E1 -8587.876,E2 -8587.876} C_VEL
LIN {X 0,Y 446.439,Z 100.496,A -85,B 0,C 180,E1 -8590.196,E2 -8590.196} C_VEL
LIN {X 0,Y 446.445,Z 100.495,A -85,B 0,C 180,E1 -8593.609,E2 -8593.609} C_VEL
LIN {X 0,Y 446.461,Z 100.496,A -85,B 0,C 180,E1 -8596.393,E2 -8596.393} C_VEL
LIN {X 0,Y 446.441,Z 100.495,A -85,B 0,C 180,E1 -8599.807,E2 -8599.807} C_VEL
LIN {X 0,Y 446.408,Z 100.502,A -85,B 0,C 180,E1 -8602.126,E2 -8602.126} C_VEL
LIN {X 0,Y 446.403,Z 100.5,A -85,B 0,C 180,E1 -8605.48,E2 -8605.48} C_VEL
LIN {X 0,Y 446.405,Z 100.503,A -85,B 0,C 180,E1 -8608.704,E2 -8608.704} C_VEL
LIN {X 0,Y 446.46,Z 100.496,A -85,B 0,C 180,E1 -8611.824,E2 -8611.824} C_VEL
LIN {X 0,Y 446.458,Z 100.494,A -85,B 0,C 180,E1 -8614.852,E2 -8614.852} C_VEL
LIN {X 0,Y 446.464,Z 100.497,A -85,B 0,C 180,E1 -8618.236,E2 -8618.236} C_VEL
LIN {X 0,Y 446.439,Z 100.5,A -85,B 0,C 180,E1 -8621.652,E2 -8621.652} C_VEL
LIN {X 0,Y 446.498,Z 100.489,A -85,B 0,C 180,E1 -8624.483,E2 -8624.483} C_VEL
LIN {X 0,Y 446.524,Z 100.487,A -85,B 0,C 180,E1 -8628.197,E2 -8628.197} C_VEL
LIN {X 0,Y 446.586,Z 100.481,A -85,B 0,C 180,E1 -8631.861,E2 -8631.861} C_VEL
LIN {X 0,Y 446.637,Z 100.471,A -85,B 0,C 180,E1 -8634.586,E2 -8634.586} C_VEL
LIN {X 0,Y 446.699,Z 100.469,A -85,B 0,C 180,E1 -8637.298,E2 -8637.298} C_VEL
LIN {X 0,Y 446.784,Z 100.453,A -85,B 0,C 180,E1 -8640.003,E2 -8640.003} C_VEL
LIN {X 0,Y 446.7,Z 100.464,A -85,B 0,C 180,E1 -8642.708,E2 -8642.708} C_VEL
LIN {X 0,Y 446.638,Z 100.471,A -85,B 0,C 180,E1 -8646.327,E2 -8646.327} C_VEL
LIN {X 0,Y 446.53,Z 100.492,A -85,B 0,C 180,E1 -8649.058,E2 -8649.058} C_VEL
LIN {X 0,Y 446.514,Z 100.491,A -85,B 0,C 180,E1 -8652.733,E2 -8652.733} C_VEL
LIN {X 0,Y 446.49,Z 100.49,A -85,B 0,C 180,E1 -8656.231,E2 -8656.231} C_VEL
LIN {X 0,Y 446.464,Z 100.494,A -85,B 0,C 180,E1 -8659.306,E2 -8659.306} C_VEL
LIN {X 0,Y 446.414,Z 100.501,A -85,B 0,C 180,E1 -8662.202,E2 -8662.202} C_VEL
LIN {X 0,Y 446.455,Z 100.495,A -85,B 0,C 180,E1 -8665.155,E2 -8665.155} C_VEL
LIN {X 0,Y 446.482,Z 100.494,A -85,B 0,C 180,E1 -8668.181,E2 -8668.181} C_VEL
LIN {X 0,Y 446.416,Z 100.5,A -85,B 0,C 180,E1 -8671.777,E2 -8671.777} C_VEL
LIN {X 0,Y 446.429,Z 100.501,A -85,B 0,C 180,E1 -8674.525,E2 -8674.525} C_VEL
LIN {X 0,Y 446.414,Z 100.505,A -85,B 0,C 180,E1 -8678.082,E2 -8678.082} C_VEL
LIN {X 0,Y 446.426,Z 100.497,A -85,B 0,C 180,E1 -8680.92,E2 -8680.92} C_VEL
LIN {X 0,Y 446.401,Z 100.506,A -85,B 0,C 180,E1 -8683.848,E2 -8683.848} C_VEL
LIN {X 0,Y 446.397,Z 100.503,A -85,B 0,C 180,E1 -8686.406,E2 -8686.406} C_VEL
LIN {X 0,Y 446.427,Z 100.497,A -85,B 0,C 180,E1 -8689.085,E2 -8689.085} C_VEL
LIN {X 0,Y 446.408,Z 100.502,A -85,B 0,C 180,E1 -8692.123,E2 -8692.123} C_VEL
LIN {X 0,Y 446.43,Z 100.502,A -85,B 0,C 180,E1 -8695.479,E2 -8695.479} C_VEL
LIN {X 0,Y 446.417,Z 100.502,A -85,B 0,C 180,E1 -8698.701,E2 -8698.701} C_VEL
LIN {X 0,Y 446.485,Z 100.564,A -85,B 0,C 180,E1 -8701.593,E2 -8701.593} C_VEL
LIN {X 0,Y 449.587,Z 115.197,A -85,B 0,C 180,E1 -8704.318,E2 -8704.318} C_VEL
LIN {X 0,Y 449.931,Z 118.805,A -85,B 0,C 180,E1 -8704.957,E2 -8704.957} C_VEL
LIN {X 0,Y 448.834,Z 137.975,A -85,B 0,C 180,E1 -8708.17,E2 -8708.17} C_VEL
LIN {X 0,Y 448.687,Z 140.384,A -85,B 0,C 180,E1 -8708.57,E2 -8708.57} C_VEL
LIN {X 0,Y 453.012,Z 166.1,A -85,B 0,C 180,E1 -8709.188,E2 -8709.188} C_VEL
LIN {X 0,Y 451.627,Z 278.699,A -85,B 0,C 180,E1 -8711.016,E2 -8711.016} C_VEL
LIN {X 0,Y 451.161,Z 293.272,A -85,B 0,C 180,E1 -8711.437,E2 -8711.437} C_VEL
LIN {X 0,Y 450.514,Z 307.573,A -85,B 0,C 180,E1 -8712.045,E2 -8712.045} C_VEL
LIN {X 0,Y 449.909,Z 319.804,A -85,B 0,C 180,E1 -8712.736,E2 -8712.736} C_VEL
LIN {X 0,Y 449.092,Z 332.509,A -85,B 0,C 180,E1 -8713.64,E2 -8713.64} C_VEL
LIN {X 0,Y 448.347,Z 344.092,A -85,B 0,C 180,E1 -8714.663,E2 -8714.663} C_VEL
LIN {X 0,Y 447.676,Z 353.728,A -85,B 0,C 180,E1 -8715.686,E2 -8715.686} C_VEL
LIN {X 0,Y 447.038,Z 364.709,A -85,B 0,C 180,E1 -8717.093,E2 -8717.093} C_VEL
LIN {X 0,Y 446.515,Z 373.274,A -85,B 0,C 180,E1 -8718.425,E2 -8718.425} C_VEL
LIN {X 0,Y 445.984,Z 381.734,A -85,B 0,C 180,E1 -8720.019,E2 -8720.019} C_VEL
LIN {X 0,Y 445.74,Z 387.624,A -85,B 0,C 180,E1 -8721.387,E2 -8721.387} C_VEL
LIN {X 0,Y 445.583,Z 392.473,A -85,B 0,C 180,E1 -8722.752,E2 -8722.752} C_VEL
LIN {X 0,Y 445.431,Z 397.478,A -85,B 0,C 180,E1 -8724.569,E2 -8724.569} C_VEL
LIN {X 0,Y 445.348,Z 400.97,A -85,B 0,C 180,E1 -8726.382,E2 -8726.382} C_VEL
LIN {X 0,Y 445.426,Z 402.187,A -85,B 0,C 180,E1 -8727.288,E2 -8727.288} C_VEL
LIN {X 0,Y 445.339,Z 403.589,A -85,B 0,C 180,E1 -8729.097,E2 -8729.097} C_VEL
LIN {X 0,Y 445.339,Z 403.652,A -85,B 0,C 180,E1 -8730.906,E2 -8730.906} C_VEL
LIN {X 0,Y 445.426,Z 402.376,A -85,B 0,C 180,E1 -8732.714,E2 -8732.714} C_VEL
LIN {X 0,Y 445.392,Z 399.723,A -85,B 0,C 180,E1 -8734.526,E2 -8734.526} C_VEL
LIN {X 0,Y 445.497,Z 395.633,A -85,B 0,C 180,E1 -8736.341,E2 -8736.341} C_VEL
LIN {X 0,Y 445.689,Z 389.993,A -85,B 0,C 180,E1 -8738.16,E2 -8738.16} C_VEL
LIN {X 0,Y 446.013,Z 383.646,A -85,B 0,C 180,E1 -8739.754,E2 -8739.754} C_VEL
LIN {X 0,Y 446.489,Z 375.764,A -85,B 0,C 180,E1 -8741.349,E2 -8741.349} C_VEL
LIN {X 0,Y 447.029,Z 367.544,A -85,B 0,C 180,E1 -8742.716,E2 -8742.716} C_VEL
LIN {X 0,Y 447.718,Z 357.661,A -85,B 0,C 180,E1 -8744.083,E2 -8744.083} C_VEL
LIN {X 0,Y 448.524,Z 346.697,A -85,B 0,C 180,E1 -8745.334,E2 -8745.334} C_VEL
LIN {X 0,Y 449.485,Z 334.531,A -85,B 0,C 180,E1 -8746.464,E2 -8746.464} C_VEL
LIN {X 0,Y 450.309,Z 321.923,A -85,B 0,C 180,E1 -8747.407,E2 -8747.407} C_VEL
LIN {X 0,Y 451.085,Z 309.241,A -85,B 0,C 180,E1 -8748.157,E2 -8748.157} C_VEL
LIN {X 0,Y 451.747,Z 295.507,A -85,B 0,C 180,E1 -8748.776,E2 -8748.776} C_VEL
LIN {X 0,Y 452.328,Z 281.262,A -85,B 0,C 180,E1 -8749.221,E2 -8749.221} C_VEL
LIN {X 0,Y 452.736,Z 261.581,A -85,B 0,C 180,E1 -8749.586,E2 -8749.586} C_VEL
LIN {X 0,Y 453.885,Z 164.742,A -85,B 0,C 180,E1 -8751.169,E2 -8751.169} C_VEL
LIN {X 0,Y 449.609,Z 142.268,A -85,B 0,C 180,E1 -8751.791,E2 -8751.791} C_VEL
LIN {X 0,Y 449.174,Z 140.004,A -85,B 0,C 180,E1 -8751.868,E2 -8751.868} C_VEL
LIN {X 0,Y 450.488,Z 120.683,A -85,B 0,C 180,E1 -8755.194,E2 -8755.194} C_VEL
LIN {X 0,Y 450.404,Z 117.961,A -85,B 0,C 180,E1 -8755.688,E2 -8755.688} C_VEL
LIN {X 0,Y 447.737,Z 105.745,A -85,B 0,C 180,E1 -8758.094,E2 -8758.094} C_VEL
LIN {X 0,Y 446.501,Z 100.493,A -85,B 0,C 180,E1 -8759.207,E2 -8759.207} C_VEL
LIN {X 0,Y 446.432,Z 100.502,A -85,B 0,C 180,E1 -8762.362,E2 -8762.362} C_VEL
LIN {X 0,Y 446.428,Z 100.502,A -85,B 0,C 180,E1 -8765.627,E2 -8765.627} C_VEL
LIN {X 0,Y 446.422,Z 100.501,A -85,B 0,C 180,E1 -8769.031,E2 -8769.031} C_VEL
LIN {X 0,Y 446.434,Z 100.501,A -85,B 0,C 180,E1 -8772.275,E2 -8772.275} C_VEL
LIN {X 0,Y 446.464,Z 100.494,A -85,B 0,C 180,E1 -8775.104,E2 -8775.104} C_VEL
LIN {X 0,Y 446.438,Z 100.485,A -85,B 0,C 180,E1 -8778.608,E2 -8778.608} C_VEL
LIN {X 0,Y 446.418,Z 100.499,A -85,B 0,C 180,E1 -8782.12,E2 -8782.12} C_VEL
LIN {X 0,Y 446.436,Z 100.499,A -85,B 0,C 180,E1 -8785.475,E2 -8785.475} C_VEL
LIN {X 0,Y 446.428,Z 100.497,A -85,B 0,C 180,E1 -8788.698,E2 -8788.698} C_VEL
LIN {X 0,Y 446.462,Z 100.491,A -85,B 0,C 180,E1 -8791.829,E2 -8791.829} C_VEL
LIN {X 0,Y 446.456,Z 100.499,A -85,B 0,C 180,E1 -8794.845,E2 -8794.845} C_VEL
LIN {X 0,Y 446.462,Z 100.495,A -85,B 0,C 180,E1 -8798.243,E2 -8798.243} C_VEL
LIN {X 0,Y 446.463,Z 100.494,A -85,B 0,C 180,E1 -8801.647,E2 -8801.647} C_VEL
LIN {X 0,Y 446.518,Z 100.485,A -85,B 0,C 180,E1 -8804.478,E2 -8804.478} C_VEL
LIN {X 0,Y 446.528,Z 100.485,A -85,B 0,C 180,E1 -8808.191,E2 -8808.191} C_VEL
LIN {X 0,Y 446.542,Z 100.485,A -85,B 0,C 180,E1 -8810.942,E2 -8810.942} C_VEL
LIN {X 0,Y 446.621,Z 100.472,A -85,B 0,C 180,E1 -8813.673,E2 -8813.673} C_VEL
LIN {X 0,Y 446.69,Z 100.461,A -85,B 0,C 180,E1 -8817.292,E2 -8817.292} C_VEL
LIN {X 0,Y 446.796,Z 100.457,A -85,B 0,C 180,E1 -8819.997,E2 -8819.997} C_VEL
LIN {X 0,Y 446.688,Z 100.467,A -85,B 0,C 180,E1 -8822.702,E2 -8822.702} C_VEL
LIN {X 0,Y 446.623,Z 100.476,A -85,B 0,C 180,E1 -8826.321,E2 -8826.321} C_VEL
LIN {X 0,Y 446.523,Z 100.488,A -85,B 0,C 180,E1 -8829.967,E2 -8829.967} C_VEL
LIN {X 0,Y 446.523,Z 100.484,A -85,B 0,C 180,E1 -8832.726,E2 -8832.726} C_VEL
LIN {X 0,Y 446.488,Z 100.488,A -85,B 0,C 180,E1 -8836.455,E2 -8836.455} C_VEL
LIN {X 0,Y 446.466,Z 100.498,A -85,B 0,C 180,E1 -8839.299,E2 -8839.299} C_VEL
LIN {X 0,Y 446.413,Z 100.5,A -85,B 0,C 180,E1 -8842.196,E2 -8842.196} C_VEL
LIN {X 0,Y 446.431,Z 100.503,A -85,B 0,C 180,E1 -8845.15,E2 -8845.15} C_VEL
LIN {X 0,Y 446.477,Z 100.492,A -85,B 0,C 180,E1 -8848.175,E2 -8848.175} C_VEL
LIN {X 0,Y 446.407,Z 100.502,A -85,B 0,C 180,E1 -8851.771,E2 -8851.771} C_VEL
LIN {X 0,Y 446.41,Z 100.496,A -85,B 0,C 180,E1 -8854.52,E2 -8854.52} C_VEL
LIN {X 0,Y 446.399,Z 100.498,A -85,B 0,C 180,E1 -8858.075,E2 -8858.075} C_VEL
LIN {X 0,Y 446.41,Z 100.5,A -85,B 0,C 180,E1 -8860.914,E2 -8860.914} C_VEL
LIN {X 0,Y 446.381,Z 100.508,A -85,B 0,C 180,E1 -8863.842,E2 -8863.842} C_VEL
LIN {X 0,Y 446.378,Z 100.514,A -85,B 0,C 180,E1 -8866.4,E2 -8866.4} C_VEL
LIN {X 0,Y 446.432,Z 100.515,A -85,B 0,C 180,E1 -8868.332,E2 -8868.332} C_VEL
LIN {X 0,Y 449.137,Z 112.962,A -85,B 0,C 180,E1 -8871.106,E2 -8871.106} C_VEL
LIN {X 0,Y 449.6,Z 117.454,A -85,B 0,C 180,E1 -8872.051,E2 -8872.051} C_VEL
LIN {X 0,Y 449.547,Z 118.285,A -85,B 0,C 180,E1 -8872.216,E2 -8872.216} C_VEL
LIN {X 0,Y 454.236,Z 138.481,A -85,B 0,C 180,E1 -8872.83,E2 -8872.83} C_VEL
LIN {X 0,Y 452.657,Z 254.939,A -85,B 0,C 180,E1 -8874.749,E2 -8874.749} C_VEL
LIN {X 0,Y 452.233,Z 269.229,A -85,B 0,C 180,E1 -8875.166,E2 -8875.166} C_VEL
LIN {X 0,Y 451.687,Z 282.621,A -85,B 0,C 180,E1 -8875.734,E2 -8875.734} C_VEL
LIN {X 0,Y 451.015,Z 294.811,A -85,B 0,C 180,E1 -8876.413,E2 -8876.413} C_VEL
LIN {X 0,Y 450.166,Z 308.093,A -85,B 0,C 180,E1 -8877.36,E2 -8877.36} C_VEL
LIN {X 0,Y 449.342,Z 319.811,A -85,B 0,C 180,E1 -8878.4,E2 -8878.4} C_VEL
LIN {X 0,Y 448.503,Z 330.975,A -85,B 0,C 180,E1 -8879.612,E2 -8879.612} C_VEL
LIN {X 0,Y 447.76,Z 340.644,A -85,B 0,C 180,E1 -8880.883,E2 -8880.883} C_VEL
LIN {X 0,Y 447.084,Z 349.201,A -85,B 0,C 180,E1 -8882.235,E2 -8882.235} C_VEL
LIN {X 0,Y 446.202,Z 352.697,A -85,B 0,C 180,E1 -8882.836,E2 -8882.836} C_VEL
LIN {X 0,Y 443.002,Z 358.078,A -85,B 0,C 180,E1 -8883.828,E2 -8883.828} C_VEL
LIN {X 0,Y 439.809,Z 362.874,A -85,B 0,C 180,E1 -8884.878,E2 -8884.878} C_VEL
LIN {X 0,Y 438.952,Z 365.456,A -85,B 0,C 180,E1 -8885.564,E2 -8885.564} C_VEL
LIN {X 0,Y 438.669,Z 371.047,A -85,B 0,C 180,E1 -8887.385,E2 -8887.385} C_VEL
LIN {X 0,Y 438.555,Z 373.443,A -85,B 0,C 180,E1 -8888.37,E2 -8888.37} C_VEL
LIN {X 0,Y 438.287,Z 376.985,A -85,B 0,C 180,E1 -8890.32,E2 -8890.32} C_VEL
LIN {X 0,Y 438.235,Z 378.158,A -85,B 0,C 180,E1 -8891.291,E2 -8891.291} C_VEL
LIN {X 0,Y 438.152,Z 379.372,A -85,B 0,C 180,E1 -8893.217,E2 -8893.217} C_VEL
LIN {X 0,Y 438.179,Z 379.158,A -85,B 0,C 180,E1 -8895.129,E2 -8895.129} C_VEL
LIN {X 0,Y 438.206,Z 377.546,A -85,B 0,C 180,E1 -8897.023,E2 -8897.023} C_VEL
LIN {X 0,Y 438.38,Z 374.52,A -85,B 0,C 180,E1 -8898.907,E2 -8898.907} C_VEL
LIN {X 0,Y 438.556,Z 370.033,A -85,B 0,C 180,E1 -8900.777,E2 -8900.777} C_VEL
LIN {X 0,Y 438.813,Z 365.574,A -85,B 0,C 180,E1 -8902.174,E2 -8902.174} C_VEL
LIN {X 0,Y 439.164,Z 359.151,A -85,B 0,C 180,E1 -8903.797,E2 -8903.797} C_VEL
LIN {X 0,Y 439.644,Z 351.196,A -85,B 0,C 180,E1 -8905.414,E2 -8905.414} C_VEL
LIN {X 0,Y 440.287,Z 342.87,A -85,B 0,C 180,E1 -8906.796,E2 -8906.796} C_VEL
LIN {X 0,Y 441.015,Z 332.879,A -85,B 0,C 180,E1 -8908.172,E2 -8908.172} C_VEL
LIN {X 0,Y 441.791,Z 321.759,A -85,B 0,C 180,E1 -8909.429,E2 -8909.429} C_VEL
LIN {X 0,Y 442.497,Z 310.73,A -85,B 0,C 180,E1 -8910.454,E2 -8910.454} C_VEL
LIN {X 0,Y 443.357,Z 297.845,A -85,B 0,C 180,E1 -8911.417,E2 -8911.417} C_VEL
LIN {X 0,Y 444.045,Z 284.342,A -85,B 0,C 180,E1 -8912.21,E2 -8912.21} C_VEL
LIN {X 0,Y 444.558,Z 270.231,A -85,B 0,C 180,E1 -8912.83,E2 -8912.83} C_VEL
LIN {X 0,Y 444.918,Z 256.317,A -85,B 0,C 180,E1 -8913.253,E2 -8913.253} C_VEL
LIN {X 0,Y 445.289,Z 226.162,A -85,B 0,C 180,E1 -8913.78,E2 -8913.78} C_VEL
LIN {X 0,Y 446.491,Z 139.431,A -85,B 0,C 180,E1 -8915.187,E2 -8915.187} C_VEL
LIN {X 0,Y 442.069,Z 118.116,A -85,B 0,C 180,E1 -8915.758,E2 -8915.758} C_VEL
LIN {X 0,Y 442.191,Z 114.918,A -85,B 0,C 180,E1 -8916.386,E2 -8916.386} C_VEL
LIN {X 0,Y 439.511,Z 101.365,A -85,B 0,C 180,E1 -8919.258,E2 -8919.258} C_VEL
LIN {X 0,Y 439.511,Z 101.367,A -85,B 0,C 180,E1 -8922.935,E2 -8922.935} C_VEL
LIN {X 0,Y 439.425,Z 101.37,A -85,B 0,C 180,E1 -8926.356,E2 -8926.356} C_VEL
LIN {X 0,Y 439.398,Z 101.379,A -85,B 0,C 180,E1 -8929.625,E2 -8929.625} C_VEL
LIN {X 0,Y 439.349,Z 101.379,A -85,B 0,C 180,E1 -8932.575,E2 -8932.575} C_VEL
LIN {X 0,Y 439.379,Z 101.38,A -85,B 0,C 180,E1 -8935.585,E2 -8935.585} C_VEL
LIN {X 0,Y 439.389,Z 101.375,A -85,B 0,C 180,E1 -8938.674,E2 -8938.674} C_VEL
LIN {X 0,Y 439.351,Z 101.378,A -85,B 0,C 180,E1 -8942.035,E2 -8942.035} C_VEL
LIN {X 0,Y 439.372,Z 101.38,A -85,B 0,C 180,E1 -8945.344,E2 -8945.344} C_VEL
LIN {X 0,Y 439.406,Z 101.375,A -85,B 0,C 180,E1 -8948.591,E2 -8948.591} C_VEL
LIN {X 0,Y 439.375,Z 101.378,A -85,B 0,C 180,E1 -8951.262,E2 -8951.262} C_VEL
LIN {X 0,Y 439.417,Z 101.377,A -85,B 0,C 180,E1 -8954.725,E2 -8954.725} C_VEL
LIN {X 0,Y 439.387,Z 101.374,A -85,B 0,C 180,E1 -8957.8,E2 -8957.8} C_VEL
LIN {X 0,Y 439.425,Z 101.372,A -85,B 0,C 180,E1 -8960.233,E2 -8960.233} C_VEL
LIN {X 0,Y 439.35,Z 101.379,A -85,B 0,C 180,E1 -8963.716,E2 -8963.716} C_VEL
LIN {X 0,Y 439.349,Z 101.379,A -85,B 0,C 180,E1 -8967.057,E2 -8967.057} C_VEL
LIN {X 0,Y 439.372,Z 101.383,A -85,B 0,C 180,E1 -8970.278,E2 -8970.278} C_VEL
LIN {X 0,Y 439.421,Z 101.371,A -85,B 0,C 180,E1 -8973.589,E2 -8973.589} C_VEL
LIN {X 0,Y 439.379,Z 101.378,A -85,B 0,C 180,E1 -8976.433,E2 -8976.433} C_VEL
LIN {X 0,Y 439.399,Z 101.374,A -85,B 0,C 180,E1 -8979.402,E2 -8979.402} C_VEL
LIN {X 0,Y 439.414,Z 101.373,A -85,B 0,C 180,E1 -8982.313,E2 -8982.313} C_VEL
LIN {X 0,Y 439.434,Z 101.369,A -85,B 0,C 180,E1 -8985.177,E2 -8985.177} C_VEL
LIN {X 0,Y 439.492,Z 101.365,A -85,B 0,C 180,E1 -8988.005,E2 -8988.005} C_VEL
LIN {X 0,Y 439.534,Z 101.362,A -85,B 0,C 180,E1 -8991.729,E2 -8991.729} C_VEL
LIN {X 0,Y 439.612,Z 101.346,A -85,B 0,C 180,E1 -8994.499,E2 -8994.499} C_VEL
LIN {X 0,Y 439.625,Z 101.345,A -85,B 0,C 180,E1 -8998.171,E2 -8998.171} C_VEL
LIN {X 0,Y 439.754,Z 101.329,A -85,B 0,C 180,E1 -9000.003,E2 -9000.003} C_VEL
LIN {X 0,Y 439.647,Z 101.343,A -85,B 0,C 180,E1 -9002.752,E2 -9002.752} C_VEL
LIN {X 0,Y 439.61,Z 101.347,A -85,B 0,C 180,E1 -9006.428,E2 -9006.428} C_VEL
LIN {X 0,Y 439.492,Z 101.367,A -85,B 0,C 180,E1 -9009.204,E2 -9009.204} C_VEL
LIN {X 0,Y 439.458,Z 101.373,A -85,B 0,C 180,E1 -9012.94,E2 -9012.94} C_VEL
LIN {X 0,Y 439.441,Z 101.369,A -85,B 0,C 180,E1 -9016.352,E2 -9016.352} C_VEL
LIN {X 0,Y 439.397,Z 101.373,A -85,B 0,C 180,E1 -9019.629,E2 -9019.629} C_VEL
LIN {X 0,Y 439.361,Z 101.384,A -85,B 0,C 180,E1 -9022.578,E2 -9022.578} C_VEL
LIN {X 0,Y 439.402,Z 101.372,A -85,B 0,C 180,E1 -9025.587,E2 -9025.587} C_VEL
LIN {X 0,Y 439.415,Z 101.375,A -85,B 0,C 180,E1 -9028.676,E2 -9028.676} C_VEL
LIN {X 0,Y 439.367,Z 101.38,A -85,B 0,C 180,E1 -9032.033,E2 -9032.033} C_VEL
LIN {X 0,Y 439.394,Z 101.373,A -85,B 0,C 180,E1 -9035.343,E2 -9035.343} C_VEL
LIN {X 0,Y 439.377,Z 101.377,A -85,B 0,C 180,E1 -9038.598,E2 -9038.598} C_VEL
LIN {X 0,Y 439.388,Z 101.374,A -85,B 0,C 180,E1 -9041.259,E2 -9041.259} C_VEL
LIN {X 0,Y 439.401,Z 101.373,A -85,B 0,C 180,E1 -9044.732,E2 -9044.732} C_VEL
LIN {X 0,Y 439.396,Z 101.38,A -85,B 0,C 180,E1 -9047.798,E2 -9047.798} C_VEL
LIN {X 0,Y 439.39,Z 101.376,A -85,B 0,C 180,E1 -9050.225,E2 -9050.225} C_VEL
LIN {X 0,Y 439.375,Z 101.383,A -85,B 0,C 180,E1 -9053.715,E2 -9053.715} C_VEL
LIN {X 0,Y 439.374,Z 101.377,A -85,B 0,C 180,E1 -9057.056,E2 -9057.056} C_VEL
LIN {X 0,Y 439.42,Z 101.377,A -85,B 0,C 180,E1 -9060.805,E2 -9060.805} C_VEL
LIN {X 0,Y 439.447,Z 101.391,A -85,B 0,C 180,E1 -9061.33,E2 -9061.33} C_VEL
LIN {X 0,Y 442.555,Z 116.048,A -85,B 0,C 180,E1 -9064.107,E2 -9064.107} C_VEL
LIN {X 0,Y 443.008,Z 120.123,A -85,B 0,C 180,E1 -9064.843,E2 -9064.843} C_VEL
LIN {X 0,Y 441.866,Z 138.982,A -85,B 0,C 180,E1 -9068.053,E2 -9068.053} C_VEL
LIN {X 0,Y 441.795,Z 140.205,A -85,B 0,C 180,E1 -9068.26,E2 -9068.26} C_VEL
LIN {X 0,Y 446.266,Z 166.999,A -85,B 0,C 180,E1 -9068.912,E2 -9068.912} C_VEL
LIN {X 0,Y 444.867,Z 278.403,A -85,B 0,C 180,E1 -9070.746,E2 -9070.746} C_VEL
LIN {X 0,Y 444.361,Z 293.017,A -85,B 0,C 180,E1 -9071.173,E2 -9071.173} C_VEL
LIN {X 0,Y 443.709,Z 306.71,A -85,B 0,C 180,E1 -9071.757,E2 -9071.757} C_VEL
LIN {X 0,Y 443.089,Z 319.131,A -85,B 0,C 180,E1 -9072.462,E2 -9072.462} C_VEL
LIN {X 0,Y 442.225,Z 331.927,A -85,B 0,C 180,E1 -9073.379,E2 -9073.379} C_VEL
LIN {X 0,Y 441.469,Z 343.58,A -85,B 0,C 180,E1 -9074.418,E2 -9074.418} C_VEL
LIN {X 0,Y 440.727,Z 353.268,A -85,B 0,C 180,E1 -9075.456,E2 -9075.456} C_VEL
LIN {X 0,Y 440.053,Z 364.192,A -85,B 0,C 180,E1 -9076.87,E2 -9076.87} C_VEL
LIN {X 0,Y 439.472,Z 372.895,A -85,B 0,C 180,E1 -9078.236,E2 -9078.236} C_VEL
LIN {X 0,Y 439.009,Z 380.262,A -85,B 0,C 180,E1 -9079.626,E2 -9079.626} C_VEL
LIN {X 0,Y 438.661,Z 387.307,A -85,B 0,C 180,E1 -9081.247,E2 -9081.247} C_VEL
LIN {X 0,Y 438.503,Z 392.186,A -85,B 0,C 180,E1 -9082.635,E2 -9082.635} C_VEL
LIN {X 0,Y 438.329,Z 397.217,A -85,B 0,C 180,E1 -9084.481,E2 -9084.481} C_VEL
LIN {X 0,Y 438.252,Z 400.731,A -85,B 0,C 180,E1 -9086.324,E2 -9086.324} C_VEL
LIN {X 0,Y 438.333,Z 401.959,A -85,B 0,C 180,E1 -9087.244,E2 -9087.244} C_VEL
LIN {X 0,Y 438.253,Z 403.38,A -85,B 0,C 180,E1 -9089.082,E2 -9089.082} C_VEL
LIN {X 0,Y 438.253,Z 403.46,A -85,B 0,C 180,E1 -9090.92,E2 -9090.92} C_VEL
LIN {X 0,Y 438.333,Z 402.207,A -85,B 0,C 180,E1 -9092.758,E2 -9092.758} C_VEL
LIN {X 0,Y 438.316,Z 399.581,A -85,B 0,C 180,E1 -9094.6,E2 -9094.6} C_VEL
LIN {X 0,Y 438.428,Z 395.514,A -85,B 0,C 180,E1 -9096.444,E2 -9096.444} C_VEL
LIN {X 0,Y 438.624,Z 389.896,A -85,B 0,C 180,E1 -9098.293,E2 -9098.293} C_VEL
LIN {X 0,Y 438.974,Z 383.573,A -85,B 0,C 180,E1 -9099.912,E2 -9099.912} C_VEL
LIN {X 0,Y 439.496,Z 375.718,A -85,B 0,C 180,E1 -9101.532,E2 -9101.532} C_VEL
LIN {X 0,Y 440.139,Z 366.493,A -85,B 0,C 180,E1 -9103.082,E2 -9103.082} C_VEL
LIN {X 0,Y 440.933,Z 355.9,A -85,B 0,C 180,E1 -9104.54,E2 -9104.54} C_VEL
LIN {X 0,Y 441.837,Z 344.57,A -85,B 0,C 180,E1 -9105.808,E2 -9105.808} C_VEL
LIN {X 0,Y 442.785,Z 333.333,A -85,B 0,C 180,E1 -9106.839,E2 -9106.839} C_VEL
LIN {X 0,Y 443.621,Z 321.317,A -85,B 0,C 180,E1 -9107.742,E2 -9107.742} C_VEL
LIN {X 0,Y 444.427,Z 308.619,A -85,B 0,C 180,E1 -9108.499,E2 -9108.499} C_VEL
LIN {X 0,Y 445.141,Z 294.738,A -85,B 0,C 180,E1 -9109.125,E2 -9109.125} C_VEL
LIN {X 0,Y 445.767,Z 280.214,A -85,B 0,C 180,E1 -9109.576,E2 -9109.576} C_VEL
LIN {X 0,Y 446.238,Z 256.555,A -85,B 0,C 180,E1 -9110.004,E2 -9110.004} C_VEL
LIN {X 0,Y 447.335,Z 165.629,A -85,B 0,C 180,E1 -9111.514,E2 -9111.514} C_VEL
LIN {X 0,Y 443.013,Z 142.831,A -85,B 0,C 180,E1 -9112.162,E2 -9112.162} C_VEL
LIN {X 0,Y 442.38,Z 139.699,A -85,B 0,C 180,E1 -9112.282,E2 -9112.282} C_VEL
LIN {X 0,Y 443.689,Z 121.6,A -85,B 0,C 180,E1 -9115.459,E2 -9115.459} C_VEL
LIN {X 0,Y 442.711,Z 115.446,A -85,B 0,C 180,E1 -9116.649,E2 -9116.649} C_VEL
LIN {X 0,Y 439.88,Z 103.165,A -85,B 0,C 180,E1 -9119.164,E2 -9119.164} C_VEL
LIN {X 0,Y 439.42,Z 101.378,A -85,B 0,C 180,E1 -9119.592,E2 -9119.592} C_VEL
LIN {X 0,Y 439.384,Z 101.383,A -85,B 0,C 180,E1 -9122.946,E2 -9122.946} C_VEL
LIN {X 0,Y 439.384,Z 101.382,A -85,B 0,C 180,E1 -9126.288,E2 -9126.288} C_VEL
LIN {X 0,Y 439.39,Z 101.376,A -85,B 0,C 180,E1 -9129.845,E2 -9129.845} C_VEL
LIN {X 0,Y 439.383,Z 101.377,A -85,B 0,C 180,E1 -9132.625,E2 -9132.625} C_VEL
LIN {X 0,Y 439.412,Z 101.374,A -85,B 0,C 180,E1 -9135.27,E2 -9135.27} C_VEL
LIN {X 0,Y 439.399,Z 101.361,A -85,B 0,C 180,E1 -9138.743,E2 -9138.743} C_VEL
LIN {X 0,Y 439.378,Z 101.382,A -85,B 0,C 180,E1 -9141.609,E2 -9141.609} C_VEL
LIN {X 0,Y 439.409,Z 101.374,A -85,B 0,C 180,E1 -9144.843,E2 -9144.843} C_VEL
LIN {X 0,Y 439.385,Z 101.374,A -85,B 0,C 180,E1 -9148.138,E2 -9148.138} C_VEL
LIN {X 0,Y 439.417,Z 101.37,A -85,B 0,C 180,E1 -9151.604,E2 -9151.604} C_VEL
LIN {X 0,Y 439.393,Z 101.375,A -85,B 0,C 180,E1 -9154.412,E2 -9154.412} C_VEL
LIN {X 0,Y 439.377,Z 101.379,A -85,B 0,C 180,E1 -9157.423,E2 -9157.423} C_VEL
LIN {X 0,Y 439.454,Z 101.365,A -85,B 0,C 180,E1 -9160.661,E2 -9160.661} C_VEL
LIN {X 0,Y 439.474,Z 101.361,A -85,B 0,C 180,E1 -9164.222,E2 -9164.222} C_VEL
LIN {X 0,Y 439.495,Z 101.36,A -85,B 0,C 180,E1 -9167.999,E2 -9167.999} C_VEL
LIN {X 0,Y 439.514,Z 101.358,A -85,B 0,C 180,E1 -9171.723,E2 -9171.723} C_VEL
LIN {X 0,Y 439.613,Z 101.353,A -85,B 0,C 180,E1 -9174.493,E2 -9174.493} C_VEL
LIN {X 0,Y 439.639,Z 101.346,A -85,B 0,C 180,E1 -9178.165,E2 -9178.165} C_VEL
LIN {X 0,Y 439.766,Z 101.332,A -85,B 0,C 180,E1 -9179.997,E2 -9179.997} C_VEL
LIN {X 0,Y 439.638,Z 101.345,A -85,B 0,C 180,E1 -9182.746,E2 -9182.746} C_VEL
LIN {X 0,Y 439.595,Z 101.351,A -85,B 0,C 180,E1 -9186.422,E2 -9186.422} C_VEL
LIN {X 0,Y 439.499,Z 101.36,A -85,B 0,C 180,E1 -9189.198,E2 -9189.198} C_VEL
LIN {X 0,Y 439.467,Z 101.363,A -85,B 0,C 180,E1 -9192.934,E2 -9192.934} C_VEL
LIN {X 0,Y 439.446,Z 101.365,A -85,B 0,C 180,E1 -9196.344,E2 -9196.344} C_VEL
LIN {X 0,Y 439.399,Z 101.374,A -85,B 0,C 180,E1 -9199.622,E2 -9199.622} C_VEL
LIN {X 0,Y 439.359,Z 101.38,A -85,B 0,C 180,E1 -9202.572,E2 -9202.572} C_VEL
LIN {X 0,Y 439.38,Z 101.376,A -85,B 0,C 180,E1 -9205.582,E2 -9205.582} C_VEL
LIN {X 0,Y 439.409,Z 101.374,A -85,B 0,C 180,E1 -9208.67,E2 -9208.67} C_VEL
LIN {X 0,Y 439.358,Z 101.38,A -85,B 0,C 180,E1 -9212.026,E2 -9212.026} C_VEL
LIN {X 0,Y 439.379,Z 101.38,A -85,B 0,C 180,E1 -9215.336,E2 -9215.336} C_VEL
LIN {X 0,Y 439.362,Z 101.378,A -85,B 0,C 180,E1 -9218.592,E2 -9218.592} C_VEL
LIN {X 0,Y 439.372,Z 101.377,A -85,B 0,C 180,E1 -9221.253,E2 -9221.253} C_VEL
LIN {X 0,Y 439.38,Z 101.381,A -85,B 0,C 180,E1 -9224.726,E2 -9224.726} C_VEL
LIN {X 0,Y 439.38,Z 101.505,A -85,B 0,C 180,E1 -9227.998,E2 -9227.998} C_VEL
LIN {X 0,Y 441.801,Z 112.355,A -85,B 0,C 180,E1 -9230.482,E2 -9230.482} C_VEL
LIN {X 0,Y 442.785,Z 118.44,A -85,B 0,C 180,E1 -9231.81,E2 -9231.81} C_VEL
LIN {X 0,Y 447.486,Z 138.342,A -85,B 0,C 180,E1 -9232.448,E2 -9232.448} C_VEL
LIN {X 0,Y 447.741,Z 143.661,A -85,B 0,C 180,E1 -9232.555,E2 -9232.555} C_VEL
LIN {X 0,Y 446.085,Z 254.708,A -85,B 0,C 180,E1 -9234.406,E2 -9234.406} C_VEL
LIN {X 0,Y 445.659,Z 268.795,A -85,B 0,C 180,E1 -9234.815,E2 -9234.815} C_VEL
LIN {X 0,Y 445.029,Z 282.951,A -85,B 0,C 180,E1 -9235.42,E2 -9235.42} C_VEL
LIN {X 0,Y 444.319,Z 295.155,A -85,B 0,C 180,E1 -9236.111,E2 -9236.111} C_VEL
LIN {X 0,Y 443.472,Z 308.057,A -85,B 0,C 180,E1 -9237.043,E2 -9237.043} C_VEL
LIN {X 0,Y 442.544,Z 320.085,A -85,B 0,C 180,E1 -9238.126,E2 -9238.126} C_VEL
LIN {X 0,Y 441.638,Z 331.482,A -85,B 0,C 180,E1 -9239.386,E2 -9239.386} C_VEL
LIN {X 0,Y 440.864,Z 340.868,A -85,B 0,C 180,E1 -9240.645,E2 -9240.645} C_VEL
LIN {X 0,Y 440.078,Z 350.183,A -85,B 0,C 180,E1 -9242.151,E2 -9242.151} C_VEL
LIN {X 0,Y 439.546,Z 357.281,A -85,B 0,C 180,E1 -9243.549,E2 -9243.549} C_VEL
LIN {X 0,Y 439.118,Z 363.015,A -85,B 0,C 180,E1 -9244.903,E2 -9244.903} C_VEL
LIN {X 0,Y 438.952,Z 365.456,A -85,B 0,C 180,E1 -9245.564,E2 -9245.564} C_VEL
LIN {X 0,Y 438.125,Z 367.871,A -85,B 0,C 180,E1 -9246.264,E2 -9246.264} C_VEL
LIN {X 0,Y 433.725,Z 372.663,A -85,B 0,C 180,E1 -9247.879,E2 -9247.879} C_VEL
LIN {X 0,Y 431.666,Z 374.864,A -85,B 0,C 180,E1 -9248.852,E2 -9248.852} C_VEL
LIN {X 0,Y 431.287,Z 375.763,A -85,B 0,C 180,E1 -9249.36,E2 -9249.36} C_VEL
LIN {X 0,Y 431.145,Z 378.081,A -85,B 0,C 180,E1 -9250.972,E2 -9250.972} C_VEL
LIN {X 0,Y 431.075,Z 379.512,A -85,B 0,C 180,E1 -9252.933,E2 -9252.933} C_VEL
LIN {X 0,Y 431.073,Z 379.478,A -85,B 0,C 180,E1 -9254.878,E2 -9254.878} C_VEL
LIN {X 0,Y 431.091,Z 378.026,A -85,B 0,C 180,E1 -9256.805,E2 -9256.805} C_VEL
LIN {X 0,Y 431.271,Z 375.161,A -85,B 0,C 180,E1 -9258.722,E2 -9258.722} C_VEL
LIN {X 0,Y 431.468,Z 370.841,A -85,B 0,C 180,E1 -9260.624,E2 -9260.624} C_VEL
LIN {X 0,Y 431.79,Z 364.945,A -85,B 0,C 180,E1 -9262.517,E2 -9262.517} C_VEL
LIN {X 0,Y 432.133,Z 358.328,A -85,B 0,C 180,E1 -9264.165,E2 -9264.165} C_VEL
LIN {X 0,Y 432.742,Z 350.085,A -85,B 0,C 180,E1 -9265.808,E2 -9265.808} C_VEL
LIN {X 0,Y 433.431,Z 341.491,A -85,B 0,C 180,E1 -9267.21,E2 -9267.21} C_VEL
LIN {X 0,Y 434.18,Z 331.119,A -85,B 0,C 180,E1 -9268.607,E2 -9268.607} C_VEL
LIN {X 0,Y 435.052,Z 319.526,A -85,B 0,C 180,E1 -9269.883,E2 -9269.883} C_VEL
LIN {X 0,Y 435.842,Z 307.957,A -85,B 0,C 180,E1 -9270.923,E2 -9270.923} C_VEL
LIN {X 0,Y 436.665,Z 295.237,A -85,B 0,C 180,E1 -9271.843,E2 -9271.843} C_VEL
LIN {X 0,Y 437.322,Z 282.093,A -85,B 0,C 180,E1 -9272.589,E2 -9272.589} C_VEL
LIN {X 0,Y 437.879,Z 267.816,A -85,B 0,C 180,E1 -9273.19,E2 -9273.19} C_VEL
LIN {X 0,Y 438.216,Z 253.544,A -85,B 0,C 180,E1 -9273.59,E2 -9273.59} C_VEL
LIN {X 0,Y 439.662,Z 139.898,A -85,B 0,C 180,E1 -9275.486,E2 -9275.486} C_VEL
LIN {X 0,Y 435.197,Z 118.274,A -85,B 0,C 180,E1 -9276.077,E2 -9276.077} C_VEL
LIN {X 0,Y 435.007,Z 115.099,A -85,B 0,C 180,E1 -9276.725,E2 -9276.725} C_VEL
LIN {X 0,Y 432.466,Z 102.243,A -85,B 0,C 180,E1 -9279.528,E2 -9279.528} C_VEL
LIN {X 0,Y 432.461,Z 102.246,A -85,B 0,C 180,E1 -9283.149,E2 -9283.149} C_VEL
LIN {X 0,Y 432.406,Z 102.244,A -85,B 0,C 180,E1 -9286.493,E2 -9286.493} C_VEL
LIN {X 0,Y 432.345,Z 102.254,A -85,B 0,C 180,E1 -9289.959,E2 -9289.959} C_VEL
LIN {X 0,Y 432.299,Z 102.259,A -85,B 0,C 180,E1 -9292.964,E2 -9292.964} C_VEL
LIN {X 0,Y 432.332,Z 102.253,A -85,B 0,C 180,E1 -9296.033,E2 -9296.033} C_VEL
LIN {X 0,Y 432.317,Z 102.262,A -85,B 0,C 180,E1 -9299.188,E2 -9299.188} C_VEL
LIN {X 0,Y 432.298,Z 102.257,A -85,B 0,C 180,E1 -9302.296,E2 -9302.296} C_VEL
LIN {X 0,Y 432.314,Z 102.258,A -85,B 0,C 180,E1 -9304.678,E2 -9304.678} C_VEL
LIN {X 0,Y 432.352,Z 102.251,A -85,B 0,C 180,E1 -9308.146,E2 -9308.146} C_VEL
LIN {X 0,Y 432.343,Z 102.251,A -85,B 0,C 180,E1 -9311.794,E2 -9311.794} C_VEL
LIN {X 0,Y 432.374,Z 102.25,A -85,B 0,C 180,E1 -9314.347,E2 -9314.347} C_VEL
LIN {X 0,Y 432.345,Z 102.255,A -85,B 0,C 180,E1 -9317.01,E2 -9317.01} C_VEL
LIN {X 0,Y 432.331,Z 102.253,A -85,B 0,C 180,E1 -9319.819,E2 -9319.819} C_VEL
LIN {X 0,Y 432.29,Z 102.26,A -85,B 0,C 180,E1 -9323.026,E2 -9323.026} C_VEL
LIN {X 0,Y 432.332,Z 102.255,A -85,B 0,C 180,E1 -9325.999,E2 -9325.999} C_VEL
LIN {X 0,Y 432.37,Z 102.25,A -85,B 0,C 180,E1 -9329.747,E2 -9329.747} C_VEL
LIN {X 0,Y 432.385,Z 102.246,A -85,B 0,C 180,E1 -9333.373,E2 -9333.373} C_VEL
LIN {X 0,Y 432.359,Z 102.256,A -85,B 0,C 180,E1 -9336.027,E2 -9336.027} C_VEL
LIN {X 0,Y 432.36,Z 102.249,A -85,B 0,C 180,E1 -9339.051,E2 -9339.051} C_VEL
LIN {X 0,Y 432.36,Z 102.255,A -85,B 0,C 180,E1 -9342.014,E2 -9342.014} C_VEL
LIN {X 0,Y 432.384,Z 102.246,A -85,B 0,C 180,E1 -9344.93,E2 -9344.93} C_VEL
LIN {X 0,Y 432.465,Z 102.243,A -85,B 0,C 180,E1 -9347.807,E2 -9347.807} C_VEL
LIN {X 0,Y 432.478,Z 102.242,A -85,B 0,C 180,E1 -9351.593,E2 -9351.593} C_VEL
LIN {X 0,Y 432.588,Z 102.221,A -85,B 0,C 180,E1 -9354.409,E2 -9354.409} C_VEL
LIN {X 0,Y 432.595,Z 102.221,A -85,B 0,C 180,E1 -9358.141,E2 -9358.141} C_VEL
LIN {X 0,Y 432.724,Z 102.205,A -85,B 0,C 180,E1 -9360.003,E2 -9360.003} C_VEL
LIN {X 0,Y 432.597,Z 102.222,A -85,B 0,C 180,E1 -9362.797,E2 -9362.797} C_VEL
LIN {X 0,Y 432.564,Z 102.225,A -85,B 0,C 180,E1 -9366.533,E2 -9366.533} C_VEL
LIN {X 0,Y 432.435,Z 102.244,A -85,B 0,C 180,E1 -9369.356,E2 -9369.356} C_VEL
LIN {X 0,Y 432.424,Z 102.247,A -85,B 0,C 180,E1 -9372.806,E2 -9372.806} C_VEL
LIN {X 0,Y 432.407,Z 102.247,A -85,B 0,C 180,E1 -9376.482,E2 -9376.482} C_VEL
LIN {X 0,Y 432.334,Z 102.253,A -85,B 0,C 180,E1 -9379.963,E2 -9379.963} C_VEL
LIN {X 0,Y 432.315,Z 102.258,A -85,B 0,C 180,E1 -9382.967,E2 -9382.967} C_VEL
LIN {X 0,Y 432.361,Z 102.251,A -85,B 0,C 180,E1 -9386.035,E2 -9386.035} C_VEL
LIN {X 0,Y 432.34,Z 102.252,A -85,B 0,C 180,E1 -9389.19,E2 -9389.19} C_VEL
LIN {X 0,Y 432.321,Z 102.26,A -85,B 0,C 180,E1 -9392.446,E2 -9392.446} C_VEL
LIN {X 0,Y 432.343,Z 102.253,A -85,B 0,C 180,E1 -9395.634,E2 -9395.634} C_VEL
LIN {X 0,Y 432.346,Z 102.251,A -85,B 0,C 180,E1 -9399.346,E2 -9399.346} C_VEL
LIN {X 0,Y 432.333,Z 102.257,A -85,B 0,C 180,E1 -9401.799,E2 -9401.799} C_VEL
LIN {X 0,Y 432.334,Z 102.255,A -85,B 0,C 180,E1 -9404.35,E2 -9404.35} C_VEL
LIN {X 0,Y 432.32,Z 102.254,A -85,B 0,C 180,E1 -9407.018,E2 -9407.018} C_VEL
LIN {X 0,Y 432.335,Z 102.26,A -85,B 0,C 180,E1 -9409.823,E2 -9409.823} C_VEL
LIN {X 0,Y 432.307,Z 102.257,A -85,B 0,C 180,E1 -9413.024,E2 -9413.024} C_VEL
LIN {X 0,Y 432.361,Z 102.255,A -85,B 0,C 180,E1 -9415.999,E2 -9415.999} C_VEL
LIN {X 0,Y 432.349,Z 102.258,A -85,B 0,C 180,E1 -9419.492,E2 -9419.492} C_VEL
LIN {X 0,Y 432.441,Z 102.409,A -85,B 0,C 180,E1 -9421.096,E2 -9421.096} C_VEL
LIN {X 0,Y 435.534,Z 117.023,A -85,B 0,C 180,E1 -9423.916,E2 -9423.916} C_VEL
LIN {X 0,Y 436.098,Z 120.076,A -85,B 0,C 180,E1 -9424.488,E2 -9424.488} C_VEL
LIN {X 0,Y 435.08,Z 137.121,A -85,B 0,C 180,E1 -9427.442,E2 -9427.442} C_VEL
LIN {X 0,Y 434.926,Z 140.181,A -85,B 0,C 180,E1 -9427.945,E2 -9427.945} C_VEL
LIN {X 0,Y 439.549,Z 167.487,A -85,B 0,C 180,E1 -9428.625,E2 -9428.625} C_VEL
LIN {X 0,Y 438.093,Z 277.823,A -85,B 0,C 180,E1 -9430.467,E2 -9430.467} C_VEL
LIN {X 0,Y 437.58,Z 292.578,A -85,B 0,C 180,E1 -9430.9,E2 -9430.9} C_VEL
LIN {X 0,Y 436.85,Z 306.887,A -85,B 0,C 180,E1 -9431.519,E2 -9431.519} C_VEL
LIN {X 0,Y 436.165,Z 320.154,A -85,B 0,C 180,E1 -9432.295,E2 -9432.295} C_VEL
LIN {X 0,Y 435.264,Z 332.729,A -85,B 0,C 180,E1 -9433.226,E2 -9433.226} C_VEL
LIN {X 0,Y 434.486,Z 344.221,A -85,B 0,C 180,E1 -9434.281,E2 -9434.281} C_VEL
LIN {X 0,Y 433.659,Z 354.765,A -85,B 0,C 180,E1 -9435.453,E2 -9435.453} C_VEL
LIN {X 0,Y 432.972,Z 365.415,A -85,B 0,C 180,E1 -9436.891,E2 -9436.891} C_VEL
LIN {X 0,Y 432.401,Z 373.883,A -85,B 0,C 180,E1 -9438.279,E2 -9438.279} C_VEL
LIN {X 0,Y 431.826,Z 382.119,A -85,B 0,C 180,E1 -9439.925,E2 -9439.925} C_VEL
LIN {X 0,Y 431.506,Z 388.749,A -85,B 0,C 180,E1 -9441.572,E2 -9441.572} C_VEL
LIN {X 0,Y 431.344,Z 393.333,A -85,B 0,C 180,E1 -9442.982,E2 -9442.982} C_VEL
LIN {X 0,Y 431.235,Z 396.951,A -85,B 0,C 180,E1 -9444.39,E2 -9444.39} C_VEL
LIN {X 0,Y 431.236,Z 398.903,A -85,B 0,C 180,E1 -9445.327,E2 -9445.327} C_VEL
LIN {X 0,Y 431.227,Z 401.726,A -85,B 0,C 180,E1 -9447.199,E2 -9447.199} C_VEL
LIN {X 0,Y 431.169,Z 403.169,A -85,B 0,C 180,E1 -9449.067,E2 -9449.067} C_VEL
LIN {X 0,Y 431.17,Z 403.27,A -85,B 0,C 180,E1 -9450.935,E2 -9450.935} C_VEL
LIN {X 0,Y 431.227,Z 402.038,A -85,B 0,C 180,E1 -9452.804,E2 -9452.804} C_VEL
LIN {X 0,Y 431.24,Z 399.439,A -85,B 0,C 180,E1 -9454.675,E2 -9454.675} C_VEL
LIN {X 0,Y 431.342,Z 395.394,A -85,B 0,C 180,E1 -9456.55,E2 -9456.55} C_VEL
LIN {X 0,Y 431.575,Z 389.799,A -85,B 0,C 180,E1 -9458.429,E2 -9458.429} C_VEL
LIN {X 0,Y 431.909,Z 383.507,A -85,B 0,C 180,E1 -9460.075,E2 -9460.075} C_VEL
LIN {X 0,Y 432.517,Z 375.694,A -85,B 0,C 180,E1 -9461.72,E2 -9461.72} C_VEL
LIN {X 0,Y 433.134,Z 367.118,A -85,B 0,C 180,E1 -9463.201,E2 -9463.201} C_VEL
LIN {X 0,Y 433.886,Z 357.768,A -85,B 0,C 180,E1 -9464.542,E2 -9464.542} C_VEL
LIN {X 0,Y 434.812,Z 346.923,A -85,B 0,C 180,E1 -9465.83,E2 -9465.83} C_VEL
LIN {X 0,Y 435.886,Z 334.923,A -85,B 0,C 180,E1 -9466.993,E2 -9466.993} C_VEL
LIN {X 0,Y 436.787,Z 322.874,A -85,B 0,C 180,E1 -9467.942,E2 -9467.942} C_VEL
LIN {X 0,Y 437.664,Z 310.211,A -85,B 0,C 180,E1 -9468.734,E2 -9468.734} C_VEL
LIN {X 0,Y 438.457,Z 296.234,A -85,B 0,C 180,E1 -9469.398,E2 -9469.398} C_VEL
LIN {X 0,Y 439.096,Z 282.548,A -85,B 0,C 180,E1 -9469.855,E2 -9469.855} C_VEL
LIN {X 0,Y 439.55,Z 265.571,A -85,B 0,C 180,E1 -9470.199,E2 -9470.199} C_VEL
LIN {X 0,Y 440.866,Z 166.726,A -85,B 0,C 180,E1 -9471.866,E2 -9471.866} C_VEL
LIN {X 0,Y 436.687,Z 144.585,A -85,B 0,C 180,E1 -9472.512,E2 -9472.512} C_VEL
LIN {X 0,Y 435.611,Z 139.604,A -85,B 0,C 180,E1 -9472.678,E2 -9472.678} C_VEL
LIN {X 0,Y 436.895,Z 122.434,A -85,B 0,C 180,E1 -9475.744,E2 -9475.744} C_VEL
LIN {X 0,Y 434.367,Z 110.323,A -85,B 0,C 180,E1 -9478.211,E2 -9478.211} C_VEL
LIN {X 0,Y 432.375,Z 102.254,A -85,B 0,C 180,E1 -9479.956,E2 -9479.956} C_VEL
LIN {X 0,Y 432.327,Z 102.262,A -85,B 0,C 180,E1 -9483.555,E2 -9483.555} C_VEL
LIN {X 0,Y 432.349,Z 102.258,A -85,B 0,C 180,E1 -9485.818,E2 -9485.818} C_VEL
LIN {X 0,Y 432.315,Z 102.259,A -85,B 0,C 180,E1 -9489.348,E2 -9489.348} C_VEL
LIN {X 0,Y 432.337,Z 102.255,A -85,B 0,C 180,E1 -9491.798,E2 -9491.798} C_VEL
LIN {X 0,Y 432.348,Z 102.255,A -85,B 0,C 180,E1 -9494.347,E2 -9494.347} C_VEL
LIN {X 0,Y 432.333,Z 102.256,A -85,B 0,C 180,E1 -9497.015,E2 -9497.015} C_VEL
LIN {X 0,Y 432.328,Z 102.25,A -85,B 0,C 180,E1 -9499.823,E2 -9499.823} C_VEL
LIN {X 0,Y 432.318,Z 102.255,A -85,B 0,C 180,E1 -9503.021,E2 -9503.021} C_VEL
LIN {X 0,Y 432.347,Z 102.253,A -85,B 0,C 180,E1 -9506.001,E2 -9506.001} C_VEL
LIN {X 0,Y 432.36,Z 102.253,A -85,B 0,C 180,E1 -9509.489,E2 -9509.489} C_VEL
LIN {X 0,Y 432.357,Z 102.248,A -85,B 0,C 180,E1 -9511.873,E2 -9511.873} C_VEL
LIN {X 0,Y 432.392,Z 102.243,A -85,B 0,C 180,E1 -9515.537,E2 -9515.537} C_VEL
LIN {X 0,Y 432.363,Z 102.25,A -85,B 0,C 180,E1 -9519.044,E2 -9519.044} C_VEL
LIN {X 0,Y 432.372,Z 102.25,A -85,B 0,C 180,E1 -9522.008,E2 -9522.008} C_VEL
LIN {X 0,Y 432.405,Z 102.247,A -85,B 0,C 180,E1 -9524.924,E2 -9524.924} C_VEL
LIN {X 0,Y 432.471,Z 102.234,A -85,B 0,C 180,E1 -9527.801,E2 -9527.801} C_VEL
LIN {X 0,Y 432.474,Z 102.235,A -85,B 0,C 180,E1 -9531.587,E2 -9531.587} C_VEL
LIN {X 0,Y 432.587,Z 102.228,A -85,B 0,C 180,E1 -9534.403,E2 -9534.403} C_VEL
LIN {X 0,Y 432.609,Z 102.221,A -85,B 0,C 180,E1 -9538.135,E2 -9538.135} C_VEL
LIN {X 0,Y 432.735,Z 102.208,A -85,B 0,C 180,E1 -9539.997,E2 -9539.997} C_VEL
LIN {X 0,Y 432.59,Z 102.223,A -85,B 0,C 180,E1 -9542.79,E2 -9542.79} C_VEL
LIN {X 0,Y 432.589,Z 102.22,A -85,B 0,C 180,E1 -9545.591,E2 -9545.591} C_VEL
LIN {X 0,Y 432.468,Z 102.236,A -85,B 0,C 180,E1 -9548.407,E2 -9548.407} C_VEL
LIN {X 0,Y 432.461,Z 102.237,A -85,B 0,C 180,E1 -9552.193,E2 -9552.193} C_VEL
LIN {X 0,Y 432.429,Z 102.24,A -85,B 0,C 180,E1 -9556.035,E2 -9556.035} C_VEL
LIN {X 0,Y 432.384,Z 102.249,A -85,B 0,C 180,E1 -9559.481,E2 -9559.481} C_VEL
LIN {X 0,Y 432.312,Z 102.259,A -85,B 0,C 180,E1 -9562.96,E2 -9562.96} C_VEL
LIN {X 0,Y 432.343,Z 102.25,A -85,B 0,C 180,E1 -9566.029,E2 -9566.029} C_VEL
LIN {X 0,Y 432.334,Z 102.246,A -85,B 0,C 180,E1 -9569.183,E2 -9569.183} C_VEL
LIN {X 0,Y 432.312,Z 102.26,A -85,B 0,C 180,E1 -9572.439,E2 -9572.439} C_VEL
LIN {X 0,Y 432.33,Z 102.257,A -85,B 0,C 180,E1 -9575.627,E2 -9575.627} C_VEL
LIN {X 0,Y 432.324,Z 102.256,A -85,B 0,C 180,E1 -9578.71,E2 -9578.71} C_VEL
LIN {X 0,Y 432.316,Z 102.257,A -85,B 0,C 180,E1 -9581.793,E2 -9581.793} C_VEL
LIN {X 0,Y 432.316,Z 102.262,A -85,B 0,C 180,E1 -9584.343,E2 -9584.343} C_VEL
LIN {X 0,Y 432.331,Z 102.37,A -85,B 0,C 180,E1 -9587.623,E2 -9587.623} C_VEL
LIN {X 0,Y 434.785,Z 113.169,A -85,B 0,C 180,E1 -9590.149,E2 -9590.149} C_VEL
LIN {X 0,Y 435.887,Z 118.87,A -85,B 0,C 180,E1 -9591.402,E2 -9591.402} C_VEL
LIN {X 0,Y 439.768,Z 133.666,A -85,B 0,C 180,E1 -9591.908,E2 -9591.908} C_VEL
LIN {X 0,Y 441.296,Z 141.167,A -85,B 0,C 180,E1 -9592.133,E2 -9592.133} C_VEL
LIN {X 0,Y 439.513,Z 255.634,A -85,B 0,C 180,E1 -9594.079,E2 -9594.079} C_VEL
LIN {X 0,Y 439.013,Z 270.045,A -85,B 0,C 180,E1 -9594.516,E2 -9594.516} C_VEL
LIN {X 0,Y 438.383,Z 283.34,A -85,B 0,C 180,E1 -9595.1,E2 -9595.1} C_VEL
LIN {X 0,Y 437.528,Z 297.431,A -85,B 0,C 180,E1 -9595.929,E2 -9595.929} C_VEL
LIN {X 0,Y 436.559,Z 310.543,A -85,B 0,C 180,E1 -9596.924,E2 -9596.924} C_VEL
LIN {X 0,Y 435.676,Z 321.652,A -85,B 0,C 180,E1 -9597.972,E2 -9597.972} C_VEL
LIN {X 0,Y 434.796,Z 331.896,A -85,B 0,C 180,E1 -9599.139,E2 -9599.139} C_VEL
LIN {X 0,Y 433.993,Z 341.129,A -85,B 0,C 180,E1 -9600.401,E2 -9600.401} C_VEL
LIN {X 0,Y 433.14,Z 350.432,A -85,B 0,C 180,E1 -9601.929,E2 -9601.929} C_VEL
LIN {X 0,Y 432.586,Z 357.344,A -85,B 0,C 180,E1 -9603.313,E2 -9603.313} C_VEL
LIN {X 0,Y 432.036,Z 364.197,A -85,B 0,C 180,E1 -9604.978,E2 -9604.978} C_VEL
LIN {X 0,Y 431.718,Z 369.17,A -85,B 0,C 180,E1 -9606.493,E2 -9606.493} C_VEL
LIN {X 0,Y 431.482,Z 373.484,A -85,B 0,C 180,E1 -9608.176,E2 -9608.176} C_VEL
LIN {X 0,Y 431.287,Z 375.763,A -85,B 0,C 180,E1 -9609.36,E2 -9609.36} C_VEL
LIN {X 0,Y 430.525,Z 377.053,A -85,B 0,C 180,E1 -9610.122,E2 -9610.122} C_VEL
LIN {X 0,Y 427.544,Z 378.618,A -85,B 0,C 180,E1 -9611.368,E2 -9611.368} C_VEL
LIN {X 0,Y 425.083,Z 379.428,A -85,B 0,C 180,E1 -9612.381,E2 -9612.381} C_VEL
LIN {X 0,Y 424.052,Z 379.769,A -85,B 0,C 180,E1 -9613.168,E2 -9613.168} C_VEL
LIN {X 0,Y 423.979,Z 379.795,A -85,B 0,C 180,E1 -9613.434,E2 -9613.434} C_VEL
LIN {X 0,Y 423.988,Z 379.745,A -85,B 0,C 180,E1 -9614.619,E2 -9614.619} C_VEL
LIN {X 0,Y 423.979,Z 378.492,A -85,B 0,C 180,E1 -9616.58,E2 -9616.58} C_VEL
LIN {X 0,Y 424.169,Z 375.795,A -85,B 0,C 180,E1 -9618.53,E2 -9618.53} C_VEL
LIN {X 0,Y 424.366,Z 371.639,A -85,B 0,C 180,E1 -9620.466,E2 -9620.466} C_VEL
LIN {X 0,Y 424.698,Z 365.914,A -85,B 0,C 180,E1 -9622.391,E2 -9622.391} C_VEL
LIN {X 0,Y 425.042,Z 359.481,A -85,B 0,C 180,E1 -9624.067,E2 -9624.067} C_VEL
LIN {X 0,Y 425.643,Z 351.493,A -85,B 0,C 180,E1 -9625.738,E2 -9625.738} C_VEL
LIN {X 0,Y 426.35,Z 343.139,A -85,B 0,C 180,E1 -9627.164,E2 -9627.164} C_VEL
LIN {X 0,Y 427.126,Z 333.118,A -85,B 0,C 180,E1 -9628.584,E2 -9628.584} C_VEL
LIN {X 0,Y 427.995,Z 321.931,A -85,B 0,C 180,E1 -9629.881,E2 -9629.881} C_VEL
LIN {X 0,Y 428.767,Z 310.845,A -85,B 0,C 180,E1 -9630.938,E2 -9630.938} C_VEL
LIN {X 0,Y 429.655,Z 298.734,A -85,B 0,C 180,E1 -9631.873,E2 -9631.873} C_VEL
LIN {X 0,Y 430.326,Z 286.508,A -85,B 0,C 180,E1 -9632.631,E2 -9632.631} C_VEL
LIN {X 0,Y 430.851,Z 273.041,A -85,B 0,C 180,E1 -9633.272,E2 -9633.272} C_VEL
LIN {X 0,Y 431.292,Z 259.175,A -85,B 0,C 180,E1 -9633.736,E2 -9633.736} C_VEL
LIN {X 0,Y 431.647,Z 240.163,A -85,B 0,C 180,E1 -9634.113,E2 -9634.113} C_VEL
LIN {X 0,Y 432.994,Z 141.029,A -85,B 0,C 180,E1 -9635.773,E2 -9635.773} C_VEL
LIN {X 0,Y 428.334,Z 118.428,A -85,B 0,C 180,E1 -9636.408,E2 -9636.408} C_VEL
LIN {X 0,Y 426.157,Z 106.645,A -85,B 0,C 180,E1 -9638.964,E2 -9638.964} C_VEL
LIN {X 0,Y 425.402,Z 103.123,A -85,B 0,C 180,E1 -9639.748,E2 -9639.748} C_VEL
LIN {X 0,Y 425.446,Z 103.12,A -85,B 0,C 180,E1 -9642.957,E2 -9642.957} C_VEL
LIN {X 0,Y 425.355,Z 103.122,A -85,B 0,C 180,E1 -9646.62,E2 -9646.62} C_VEL
LIN {X 0,Y 425.325,Z 103.132,A -85,B 0,C 180,E1 -9649.649,E2 -9649.649} C_VEL
LIN {X 0,Y 425.3,Z 103.129,A -85,B 0,C 180,E1 -9652.336,E2 -9652.336} C_VEL
LIN {X 0,Y 425.266,Z 103.139,A -85,B 0,C 180,E1 -9655.446,E2 -9655.446} C_VEL
LIN {X 0,Y 425.301,Z 103.13,A -85,B 0,C 180,E1 -9658.633,E2 -9658.633} C_VEL
LIN {X 0,Y 425.24,Z 103.137,A -85,B 0,C 180,E1 -9661.927,E2 -9661.927} C_VEL
LIN {X 0,Y 425.274,Z 103.136,A -85,B 0,C 180,E1 -9665.336,E2 -9665.336} C_VEL
LIN {X 0,Y 425.318,Z 103.133,A -85,B 0,C 180,E1 -9668.894,E2 -9668.894} C_VEL
LIN {X 0,Y 425.304,Z 103.133,A -85,B 0,C 180,E1 -9672.647,E2 -9672.647} C_VEL
LIN {X 0,Y 425.324,Z 103.127,A -85,B 0,C 180,E1 -9676.059,E2 -9676.059} C_VEL
LIN {X 0,Y 425.282,Z 103.138,A -85,B 0,C 180,E1 -9678.628,E2 -9678.628} C_VEL
LIN {X 0,Y 425.298,Z 103.131,A -85,B 0,C 180,E1 -9681.107,E2 -9681.107} C_VEL
LIN {X 0,Y 425.273,Z 103.137,A -85,B 0,C 180,E1 -9684.667,E2 -9684.667} C_VEL
LIN {X 0,Y 425.248,Z 103.139,A -85,B 0,C 180,E1 -9688.077,E2 -9688.077} C_VEL
LIN {X 0,Y 425.313,Z 103.127,A -85,B 0,C 180,E1 -9691.371,E2 -9691.371} C_VEL
LIN {X 0,Y 425.286,Z 103.133,A -85,B 0,C 180,E1 -9694.559,E2 -9694.559} C_VEL
LIN {X 0,Y 425.308,Z 103.131,A -85,B 0,C 180,E1 -9697.72,E2 -9697.72} C_VEL
LIN {X 0,Y 425.356,Z 103.122,A -85,B 0,C 180,E1 -9700.708,E2 -9700.708} C_VEL
LIN {X 0,Y 425.38,Z 103.124,A -85,B 0,C 180,E1 -9703.692,E2 -9703.692} C_VEL
LIN {X 0,Y 425.414,Z 103.12,A -85,B 0,C 180,E1 -9707.602,E2 -9707.602} C_VEL
LIN {X 0,Y 425.428,Z 103.118,A -85,B 0,C 180,E1 -9711.453,E2 -9711.453} C_VEL
LIN {X 0,Y 425.544,Z 103.099,A -85,B 0,C 180,E1 -9714.316,E2 -9714.316} C_VEL
LIN {X 0,Y 425.565,Z 103.096,A -85,B 0,C 180,E1 -9718.11,E2 -9718.11} C_VEL
LIN {X 0,Y 425.694,Z 103.081,A -85,B 0,C 180,E1 -9720.003,E2 -9720.003} C_VEL
LIN {X 0,Y 425.548,Z 103.1,A -85,B 0,C 180,E1 -9722.843,E2 -9722.843} C_VEL
LIN {X 0,Y 425.522,Z 103.103,A -85,B 0,C 180,E1 -9726.642,E2 -9726.642} C_VEL
LIN {X 0,Y 425.393,Z 103.119,A -85,B 0,C 180,E1 -9729.512,E2 -9729.512} C_VEL
LIN {X 0,Y 425.386,Z 103.125,A -85,B 0,C 180,E1 -9732.907,E2 -9732.907} C_VEL
LIN {X 0,Y 425.356,Z 103.126,A -85,B 0,C 180,E1 -9736.608,E2 -9736.608} C_VEL
LIN {X 0,Y 425.324,Z 103.126,A -85,B 0,C 180,E1 -9739.639,E2 -9739.639} C_VEL
LIN {X 0,Y 425.303,Z 103.129,A -85,B 0,C 180,E1 -9743.368,E2 -9743.368} C_VEL
LIN {X 0,Y 425.346,Z 103.126,A -85,B 0,C 180,E1 -9746.847,E2 -9746.847} C_VEL
LIN {X 0,Y 425.288,Z 103.131,A -85,B 0,C 180,E1 -9749.722,E2 -9749.722} C_VEL
LIN {X 0,Y 425.28,Z 103.132,A -85,B 0,C 180,E1 -9753.051,E2 -9753.051} C_VEL
LIN {X 0,Y 425.282,Z 103.135,A -85,B 0,C 180,E1 -9755.931,E2 -9755.931} C_VEL
LIN {X 0,Y 425.292,Z 103.13,A -85,B 0,C 180,E1 -9759.045,E2 -9759.045} C_VEL
LIN {X 0,Y 425.275,Z 103.133,A -85,B 0,C 180,E1 -9762.655,E2 -9762.655} C_VEL
LIN {X 0,Y 425.262,Z 103.139,A -85,B 0,C 180,E1 -9766.046,E2 -9766.046} C_VEL
LIN {X 0,Y 425.274,Z 103.132,A -85,B 0,C 180,E1 -9768.623,E2 -9768.623} C_VEL
LIN {X 0,Y 425.293,Z 103.13,A -85,B 0,C 180,E1 -9771.103,E2 -9771.103} C_VEL
LIN {X 0,Y 425.301,Z 103.129,A -85,B 0,C 180,E1 -9774.666,E2 -9774.666} C_VEL
LIN {X 0,Y 425.266,Z 103.139,A -85,B 0,C 180,E1 -9778.075,E2 -9778.075} C_VEL
LIN {X 0,Y 425.336,Z 103.147,A -85,B 0,C 180,E1 -9780.8,E2 -9780.8} C_VEL
LIN {X 0,Y 428.551,Z 117.985,A -85,B 0,C 180,E1 -9783.72,E2 -9783.72} C_VEL
LIN {X 0,Y 429.145,Z 122.759,A -85,B 0,C 180,E1 -9784.616,E2 -9784.616} C_VEL
LIN {X 0,Y 428.01,Z 139.784,A -85,B 0,C 180,E1 -9787.606,E2 -9787.606} C_VEL
LIN {X 0,Y 432.842,Z 168.75,A -85,B 0,C 180,E1 -9788.345,E2 -9788.345} C_VEL
LIN {X 0,Y 431.304,Z 278.418,A -85,B 0,C 180,E1 -9790.208,E2 -9790.208} C_VEL
LIN {X 0,Y 430.771,Z 292.901,A -85,B 0,C 180,E1 -9790.648,E2 -9790.648} C_VEL
LIN {X 0,Y 430.044,Z 306.687,A -85,B 0,C 180,E1 -9791.257,E2 -9791.257} C_VEL
LIN {X 0,Y 429.333,Z 319.367,A -85,B 0,C 180,E1 -9792.004,E2 -9792.004} C_VEL
LIN {X 0,Y 428.413,Z 332.057,A -85,B 0,C 180,E1 -9792.95,E2 -9792.95} C_VEL
LIN {X 0,Y 427.579,Z 343.632,A -85,B 0,C 180,E1 -9794.021,E2 -9794.021} C_VEL
LIN {X 0,Y 426.707,Z 354.242,A -85,B 0,C 180,E1 -9795.211,E2 -9795.211} C_VEL
LIN {X 0,Y 425.978,Z 364.787,A -85,B 0,C 180,E1 -9796.647,E2 -9796.647} C_VEL
LIN {X 0,Y 425.358,Z 373.472,A -85,B 0,C 180,E1 -9798.082,E2 -9798.082} C_VEL
LIN {X 0,Y 424.779,Z 381.769,A -85,B 0,C 180,E1 -9799.756,E2 -9799.756} C_VEL
LIN {X 0,Y 424.442,Z 388.436,A -85,B 0,C 180,E1 -9801.431,E2 -9801.431} C_VEL
LIN {X 0,Y 424.265,Z 393.038,A -85,B 0,C 180,E1 -9802.865,E2 -9802.865} C_VEL
LIN {X 0,Y 424.144,Z 396.683,A -85,B 0,C 180,E1 -9804.296,E2 -9804.296} C_VEL
LIN {X 0,Y 424.16,Z 398.648,A -85,B 0,C 180,E1 -9805.249,E2 -9805.249} C_VEL
LIN {X 0,Y 424.123,Z 401.493,A -85,B 0,C 180,E1 -9807.152,E2 -9807.152} C_VEL
LIN {X 0,Y 424.089,Z 402.958,A -85,B 0,C 180,E1 -9809.052,E2 -9809.052} C_VEL
LIN {X 0,Y 424.089,Z 403.079,A -85,B 0,C 180,E1 -9810.951,E2 -9810.951} C_VEL
LIN {X 0,Y 424.121,Z 401.868,A -85,B 0,C 180,E1 -9812.851,E2 -9812.851} C_VEL
LIN {X 0,Y 424.166,Z 399.3,A -85,B 0,C 180,E1 -9814.753,E2 -9814.753} C_VEL
LIN {X 0,Y 424.253,Z 395.288,A -85,B 0,C 180,E1 -9816.66,E2 -9816.66} C_VEL
LIN {X 0,Y 424.501,Z 389.726,A -85,B 0,C 180,E1 -9818.57,E2 -9818.57} C_VEL
LIN {X 0,Y 424.872,Z 383.467,A -85,B 0,C 180,E1 -9820.244,E2 -9820.244} C_VEL
LIN {X 0,Y 425.546,Z 375.688,A -85,B 0,C 180,E1 -9821.915,E2 -9821.915} C_VEL
LIN {X 0,Y 426.137,Z 367.587,A -85,B 0,C 180,E1 -9823.351,E2 -9823.351} C_VEL
LIN {X 0,Y 426.985,Z 357.846,A -85,B 0,C 180,E1 -9824.782,E2 -9824.782} C_VEL
LIN {X 0,Y 427.958,Z 347.057,A -85,B 0,C 180,E1 -9826.09,E2 -9826.09} C_VEL
LIN {X 0,Y 429.104,Z 335.138,A -85,B 0,C 180,E1 -9827.27,E2 -9827.27} C_VEL
LIN {X 0,Y 430.046,Z 323.319,A -85,B 0,C 180,E1 -9828.224,E2 -9828.224} C_VEL
LIN {X 0,Y 431.049,Z 309.691,A -85,B 0,C 180,E1 -9829.095,E2 -9829.095} C_VEL
LIN {X 0,Y 431.875,Z 295.607,A -85,B 0,C 180,E1 -9829.767,E2 -9829.767} C_VEL
LIN {X 0,Y 432.576,Z 281.734,A -85,B 0,C 180,E1 -9830.229,E2 -9830.229} C_VEL
LIN {X 0,Y 433.008,Z 264.475,A -85,B 0,C 180,E1 -9830.58,E2 -9830.58} C_VEL
LIN {X 0,Y 434.43,Z 167.909,A -85,B 0,C 180,E1 -9832.23,E2 -9832.23} C_VEL
LIN {X 0,Y 430.257,Z 145.952,A -85,B 0,C 180,E1 -9832.888,E2 -9832.888} C_VEL
LIN {X 0,Y 428.846,Z 139.306,A -85,B 0,C 180,E1 -9833.124,E2 -9833.124} C_VEL
LIN {X 0,Y 430.086,Z 124.624,A -85,B 0,C 180,E1 -9835.789,E2 -9835.789} C_VEL
LIN {X 0,Y 428.027,Z 114.15,A -85,B 0,C 180,E1 -9837.947,E2 -9837.947} C_VEL
LIN {X 0,Y 425.312,Z 103.132,A -85,B 0,C 180,E1 -9840.389,E2 -9840.389} C_VEL
LIN {X 0,Y 425.283,Z 103.14,A -85,B 0,C 180,E1 -9843.049,E2 -9843.049} C_VEL
LIN {X 0,Y 425.293,Z 103.138,A -85,B 0,C 180,E1 -9845.928,E2 -9845.928} C_VEL
LIN {X 0,Y 425.275,Z 103.136,A -85,B 0,C 180,E1 -9849.037,E2 -9849.037} C_VEL
LIN {X 0,Y 425.296,Z 103.135,A -85,B 0,C 180,E1 -9851.957,E2 -9851.957} C_VEL
LIN {X 0,Y 425.299,Z 103.132,A -85,B 0,C 180,E1 -9855.283,E2 -9855.283} C_VEL
LIN {X 0,Y 425.282,Z 103.119,A -85,B 0,C 180,E1 -9858.62,E2 -9858.62} C_VEL
LIN {X 0,Y 425.294,Z 103.132,A -85,B 0,C 180,E1 -9861.099,E2 -9861.099} C_VEL
LIN {X 0,Y 425.309,Z 103.13,A -85,B 0,C 180,E1 -9864.663,E2 -9864.663} C_VEL
LIN {X 0,Y 425.278,Z 103.132,A -85,B 0,C 180,E1 -9868.072,E2 -9868.072} C_VEL
LIN {X 0,Y 425.324,Z 103.129,A -85,B 0,C 180,E1 -9871.365,E2 -9871.365} C_VEL
LIN {X 0,Y 425.286,Z 103.134,A -85,B 0,C 180,E1 -9874.552,E2 -9874.552} C_VEL
LIN {X 0,Y 425.298,Z 103.127,A -85,B 0,C 180,E1 -9876.632,E2 -9876.632} C_VEL
LIN {X 0,Y 425.308,Z 103.123,A -85,B 0,C 180,E1 -9879.693,E2 -9879.693} C_VEL
LIN {X 0,Y 425.345,Z 103.128,A -85,B 0,C 180,E1 -9882.695,E2 -9882.695} C_VEL
LIN {X 0,Y 425.358,Z 103.123,A -85,B 0,C 180,E1 -9885.648,E2 -9885.648} C_VEL
LIN {X 0,Y 425.36,Z 103.121,A -85,B 0,C 180,E1 -9888.561,E2 -9888.561} C_VEL
LIN {X 0,Y 425.418,Z 103.114,A -85,B 0,C 180,E1 -9891.447,E2 -9891.447} C_VEL
LIN {X 0,Y 425.541,Z 103.104,A -85,B 0,C 180,E1 -9894.31,E2 -9894.31} C_VEL
LIN {X 0,Y 425.578,Z 103.096,A -85,B 0,C 180,E1 -9898.104,E2 -9898.104} C_VEL
LIN {X 0,Y 425.705,Z 103.083,A -85,B 0,C 180,E1 -9899.997,E2 -9899.997} C_VEL
LIN {X 0,Y 425.543,Z 103.1,A -85,B 0,C 180,E1 -9902.837,E2 -9902.837} C_VEL
LIN {X 0,Y 425.501,Z 103.104,A -85,B 0,C 180,E1 -9906.518,E2 -9906.518} C_VEL
LIN {X 0,Y 425.401,Z 103.116,A -85,B 0,C 180,E1 -9909.506,E2 -9909.506} C_VEL
LIN {X 0,Y 425.395,Z 103.116,A -85,B 0,C 180,E1 -9912.9,E2 -9912.9} C_VEL
LIN {X 0,Y 425.36,Z 103.119,A -85,B 0,C 180,E1 -9916.601,E2 -9916.601} C_VEL
LIN {X 0,Y 425.326,Z 103.127,A -85,B 0,C 180,E1 -9919.631,E2 -9919.631} C_VEL
LIN {X 0,Y 425.284,Z 103.132,A -85,B 0,C 180,E1 -9922.335,E2 -9922.335} C_VEL
LIN {X 0,Y 425.313,Z 103.13,A -85,B 0,C 180,E1 -9924.653,E2 -9924.653} C_VEL
LIN {X 0,Y 425.338,Z 103.128,A -85,B 0,C 180,E1 -9927.554,E2 -9927.554} C_VEL
LIN {X 0,Y 425.278,Z 103.127,A -85,B 0,C 180,E1 -9930.812,E2 -9930.812} C_VEL
LIN {X 0,Y 425.298,Z 103.124,A -85,B 0,C 180,E1 -9934.283,E2 -9934.283} C_VEL
LIN {X 0,Y 425.264,Z 103.13,A -85,B 0,C 180,E1 -9937.69,E2 -9937.69} C_VEL
LIN {X 0,Y 425.263,Z 103.135,A -85,B 0,C 180,E1 -9940.516,E2 -9940.516} C_VEL
LIN {X 0,Y 425.24,Z 103.141,A -85,B 0,C 180,E1 -9943.347,E2 -9943.347} C_VEL
LIN {X 0,Y 425.236,Z 103.146,A -85,B 0,C 180,E1 -9946.646,E2 -9946.646} C_VEL
LIN {X 0,Y 425.281,Z 103.271,A -85,B 0,C 180,E1 -9947.241,E2 -9947.241} C_VEL
LIN {X 0,Y 427.963,Z 114.894,A -85,B 0,C 180,E1 -9950.012,E2 -9950.012} C_VEL
LIN {X 0,Y 428.801,Z 119.108,A -85,B 0,C 180,E1 -9950.95,E2 -9950.95} C_VEL
LIN {X 0,Y 430.997,Z 125.434,A -85,B 0,C 180,E1 -9951.21,E2 -9951.21} C_VEL
LIN {X 0,Y 434.742,Z 141.613,A -85,B 0,C 180,E1 -9951.742,E2 -9951.742} C_VEL
LIN {X 0,Y 433,Z 255.263,A -85,B 0,C 180,E1 -9953.705,E2 -9953.705} C_VEL
LIN {X 0,Y 432.523,Z 269.315,A -85,B 0,C 180,E1 -9954.127,E2 -9954.127} C_VEL
LIN {X 0,Y 431.845,Z 282.875,A -85,B 0,C 180,E1 -9954.72,E2 -9954.72} C_VEL
LIN {X 0,Y 430.99,Z 295.938,A -85,B 0,C 180,E1 -9955.481,E2 -9955.481} C_VEL
LIN {X 0,Y 430.04,Z 308.847,A -85,B 0,C 180,E1 -9956.449,E2 -9956.449} C_VEL
LIN {X 0,Y 429.015,Z 320.696,A -85,B 0,C 180,E1 -9957.553,E2 -9957.553} C_VEL
LIN {X 0,Y 428.098,Z 330.796,A -85,B 0,C 180,E1 -9958.697,E2 -9958.697} C_VEL
LIN {X 0,Y 427.12,Z 341.39,A -85,B 0,C 180,E1 -9960.148,E2 -9960.148} C_VEL
LIN {X 0,Y 426.234,Z 350.685,A -85,B 0,C 180,E1 -9961.701,E2 -9961.701} C_VEL
LIN {X 0,Y 425.626,Z 357.426,A -85,B 0,C 180,E1 -9963.071,E2 -9963.071} C_VEL
LIN {X 0,Y 425.094,Z 363.467,A -85,B 0,C 180,E1 -9964.54,E2 -9964.54} C_VEL
LIN {X 0,Y 424.71,Z 368.64,A -85,B 0,C 180,E1 -9966.081,E2 -9966.081} C_VEL
LIN {X 0,Y 424.417,Z 373.608,A -85,B 0,C 180,E1 -9968.006,E2 -9968.006} C_VEL
LIN {X 0,Y 424.168,Z 376.641,A -85,B 0,C 180,E1 -9969.637,E2 -9969.637} C_VEL
LIN {X 0,Y 424.021,Z 378.977,A -85,B 0,C 180,E1 -9971.643,E2 -9971.643} C_VEL
LIN {X 0,Y 423.979,Z 379.795,A -85,B 0,C 180,E1 -9973.434,E2 -9973.434} C_VEL
LIN {X 0,Y 423.329,Z 379.876,A -85,B 0,C 180,E1 -9974.227,E2 -9974.227} C_VEL
LIN {X 0,Y 420.446,Z 379.482,A -85,B 0,C 180,E1 -9975.515,E2 -9975.515} C_VEL
LIN {X 0,Y 418.027,Z 378.686,A -85,B 0,C 180,E1 -9976.55,E2 -9976.55} C_VEL
LIN {X 0,Y 417.038,Z 377.807,A -85,B 0,C 180,E1 -9977.345,E2 -9977.345} C_VEL
LIN {X 0,Y 416.985,Z 377.443,A -85,B 0,C 180,E1 -9977.613,E2 -9977.613} C_VEL
LIN {X 0,Y 417.168,Z 374.6,A -85,B 0,C 180,E1 -9979.319,E2 -9979.319} C_VEL
LIN {X 0,Y 417.378,Z 369.863,A -85,B 0,C 180,E1 -9981.282,E2 -9981.282} C_VEL
LIN {X 0,Y 417.741,Z 364.414,A -85,B 0,C 180,E1 -9982.985,E2 -9982.985} C_VEL
LIN {X 0,Y 418.176,Z 357.511,A -85,B 0,C 180,E1 -9984.695,E2 -9984.695} C_VEL
LIN {X 0,Y 418.847,Z 348.99,A -85,B 0,C 180,E1 -9986.391,E2 -9986.391} C_VEL
LIN {X 0,Y 419.58,Z 340.111,A -85,B 0,C 180,E1 -9987.839,E2 -9987.839} C_VEL
LIN {X 0,Y 420.467,Z 329.38,A -85,B 0,C 180,E1 -9989.28,E2 -9989.28} C_VEL
LIN {X 0,Y 421.381,Z 318.498,A -85,B 0,C 180,E1 -9990.477,E2 -9990.477} C_VEL
LIN {X 0,Y 422.166,Z 307.705,A -85,B 0,C 180,E1 -9991.457,E2 -9991.457} C_VEL
LIN {X 0,Y 423.031,Z 295.228,A -85,B 0,C 180,E1 -9992.379,E2 -9992.379} C_VEL
LIN {X 0,Y 423.73,Z 281.966,A -85,B 0,C 180,E1 -9993.148,E2 -9993.148} C_VEL
LIN {X 0,Y 424.333,Z 268.227,A -85,B 0,C 180,E1 -9993.738,E2 -9993.738} C_VEL
LIN {X 0,Y 424.654,Z 254.032,A -85,B 0,C 180,E1 -9994.151,E2 -9994.151} C_VEL
LIN {X 0,Y 426.356,Z 142.465,A -85,B 0,C 180,E1 -9996.059,E2 -9996.059} C_VEL
LIN {X 0,Y 421.289,Z 118.706,A -85,B 0,C 180,E1 -9996.735,E2 -9996.735} C_VEL
LIN {X 0,Y 418.665,Z 105.48,A -85,B 0,C 180,E1 -9999.662,E2 -9999.662} C_VEL
LIN {X 0,Y 418.317,Z 104.006,A -85,B 0,C 180,E1 -10000.037,E2 -10000.037} C_VEL
LIN {X 0,Y 418.403,Z 103.998,A -85,B 0,C 180,E1 -10003.057,E2 -10003.057} C_VEL
LIN {X 0,Y 418.303,Z 104.001,A -85,B 0,C 180,E1 -10006.748,E2 -10006.748} C_VEL
LIN {X 0,Y 418.267,Z 104.009,A -85,B 0,C 180,E1 -10009.803,E2 -10009.803} C_VEL
LIN {X 0,Y 418.253,Z 104.007,A -85,B 0,C 180,E1 -10012.734,E2 -10012.734} C_VEL
LIN {X 0,Y 418.238,Z 104.01,A -85,B 0,C 180,E1 -10015.905,E2 -10015.905} C_VEL
LIN {X 0,Y 418.239,Z 104.015,A -85,B 0,C 180,E1 -10019.162,E2 -10019.162} C_VEL
LIN {X 0,Y 418.226,Z 104.014,A -85,B 0,C 180,E1 -10022.846,E2 -10022.846} C_VEL
LIN {X 0,Y 418.229,Z 104.01,A -85,B 0,C 180,E1 -10026.243,E2 -10026.243} C_VEL
LIN {X 0,Y 418.244,Z 104.008,A -85,B 0,C 180,E1 -10029.681,E2 -10029.681} C_VEL
LIN {X 0,Y 418.256,Z 104.008,A -85,B 0,C 180,E1 -10032.332,E2 -10032.332} C_VEL
LIN {X 0,Y 418.258,Z 104.009,A -85,B 0,C 180,E1 -10035.118,E2 -10035.118} C_VEL
LIN {X 0,Y 418.266,Z 104.005,A -85,B 0,C 180,E1 -10037.776,E2 -10037.776} C_VEL
LIN {X 0,Y 418.24,Z 104.008,A -85,B 0,C 180,E1 -10041.562,E2 -10041.562} C_VEL
LIN {X 0,Y 418.232,Z 104.01,A -85,B 0,C 180,E1 -10045.162,E2 -10045.162} C_VEL
LIN {X 0,Y 418.223,Z 104.01,A -85,B 0,C 180,E1 -10047.475,E2 -10047.475} C_VEL
LIN {X 0,Y 418.252,Z 104.008,A -85,B 0,C 180,E1 -10050.896,E2 -10050.896} C_VEL
LIN {X 0,Y 418.259,Z 104.013,A -85,B 0,C 180,E1 -10054.1,E2 -10054.1} C_VEL
LIN {X 0,Y 418.276,Z 104.006,A -85,B 0,C 180,E1 -10057.533,E2 -10057.533} C_VEL
LIN {X 0,Y 418.31,Z 104.002,A -85,B 0,C 180,E1 -10060.37,E2 -10060.37} C_VEL
LIN {X 0,Y 418.307,Z 104.002,A -85,B 0,C 180,E1 -10063.408,E2 -10063.408} C_VEL
LIN {X 0,Y 418.338,Z 103.996,A -85,B 0,C 180,E1 -10066.997,E2 -10066.997} C_VEL
LIN {X 0,Y 418.346,Z 103.996,A -85,B 0,C 180,E1 -10070.332,E2 -10070.332} C_VEL
LIN {X 0,Y 418.481,Z 103.982,A -85,B 0,C 180,E1 -10073.252,E2 -10073.252} C_VEL
LIN {X 0,Y 418.333,Z 104,A -85,B 0,C 180,E1 -10075.185,E2 -10075.185} C_VEL
LIN {X 0,Y 418.534,Z 103.972,A -85,B 0,C 180,E1 -10078.079,E2 -10078.079} C_VEL
LIN {X 0,Y 418.663,Z 103.956,A -85,B 0,C 180,E1 -10080.003,E2 -10080.003} C_VEL
LIN {X 0,Y 418.502,Z 103.979,A -85,B 0,C 180,E1 -10082.891,E2 -10082.891} C_VEL
LIN {X 0,Y 418.485,Z 103.981,A -85,B 0,C 180,E1 -10086.754,E2 -10086.754} C_VEL
LIN {X 0,Y 418.334,Z 103.998,A -85,B 0,C 180,E1 -10089.674,E2 -10089.674} C_VEL
LIN {X 0,Y 418.339,Z 104.003,A -85,B 0,C 180,E1 -10093.004,E2 -10093.004} C_VEL
LIN {X 0,Y 418.307,Z 104.006,A -85,B 0,C 180,E1 -10096.738,E2 -10096.738} C_VEL
LIN {X 0,Y 418.266,Z 104.005,A -85,B 0,C 180,E1 -10099.793,E2 -10099.793} C_VEL
LIN {X 0,Y 418.234,Z 104.015,A -85,B 0,C 180,E1 -10102.739,E2 -10102.739} C_VEL
LIN {X 0,Y 418.268,Z 104.006,A -85,B 0,C 180,E1 -10105.907,E2 -10105.907} C_VEL
LIN {X 0,Y 418.262,Z 104.006,A -85,B 0,C 180,E1 -10109.165,E2 -10109.165} C_VEL
LIN {X 0,Y 418.255,Z 104.008,A -85,B 0,C 180,E1 -10112.846,E2 -10112.846} C_VEL
LIN {X 0,Y 418.244,Z 104.015,A -85,B 0,C 180,E1 -10116.241,E2 -10116.241} C_VEL
LIN {X 0,Y 418.248,Z 104.01,A -85,B 0,C 180,E1 -10119.685,E2 -10119.685} C_VEL
LIN {X 0,Y 418.229,Z 104.013,A -85,B 0,C 180,E1 -10122.324,E2 -10122.324} C_VEL
LIN {X 0,Y 418.236,Z 104.009,A -85,B 0,C 180,E1 -10125.111,E2 -10125.111} C_VEL
LIN {X 0,Y 418.24,Z 104.014,A -85,B 0,C 180,E1 -10127.769,E2 -10127.769} C_VEL
LIN {X 0,Y 418.243,Z 104.008,A -85,B 0,C 180,E1 -10130.623,E2 -10130.623} C_VEL
LIN {X 0,Y 418.244,Z 104.011,A -85,B 0,C 180,E1 -10133.978,E2 -10133.978} C_VEL
LIN {X 0,Y 418.26,Z 104.008,A -85,B 0,C 180,E1 -10137.158,E2 -10137.158} C_VEL
LIN {X 0,Y 418.282,Z 104.044,A -85,B 0,C 180,E1 -10140.531,E2 -10140.531} C_VEL
LIN {X 0,Y 421.737,Z 120.024,A -85,B 0,C 180,E1 -10143.727,E2 -10143.727} C_VEL
LIN {X 0,Y 422.265,Z 123.313,A -85,B 0,C 180,E1 -10144.361,E2 -10144.361} C_VEL
LIN {X 0,Y 421.139,Z 139.627,A -85,B 0,C 180,E1 -10147.275,E2 -10147.275} C_VEL
LIN {X 0,Y 426.129,Z 169.096,A -85,B 0,C 180,E1 -10148.041,E2 -10148.041} C_VEL
LIN {X 0,Y 424.535,Z 277.75,A -85,B 0,C 180,E1 -10149.911,E2 -10149.911} C_VEL
LIN {X 0,Y 424.007,Z 292.406,A -85,B 0,C 180,E1 -10150.358,E2 -10150.358} C_VEL
LIN {X 0,Y 423.28,Z 305.9,A -85,B 0,C 180,E1 -10150.956,E2 -10150.956} C_VEL
LIN {X 0,Y 422.523,Z 318.573,A -85,B 0,C 180,E1 -10151.704,E2 -10151.704} C_VEL
LIN {X 0,Y 421.554,Z 331.383,A -85,B 0,C 180,E1 -10152.664,E2 -10152.664} C_VEL
LIN {X 0,Y 420.662,Z 343.041,A -85,B 0,C 180,E1 -10153.751,E2 -10153.751} C_VEL
LIN {X 0,Y 419.776,Z 353.72,A -85,B 0,C 180,E1 -10154.961,E2 -10154.961} C_VEL
LIN {X 0,Y 419.002,Z 364.319,A -85,B 0,C 180,E1 -10156.42,E2 -10156.42} C_VEL
LIN {X 0,Y 418.327,Z 373.05,A -85,B 0,C 180,E1 -10157.879,E2 -10157.879} C_VEL
LIN {X 0,Y 417.741,Z 381.405,A -85,B 0,C 180,E1 -10159.582,E2 -10159.582} C_VEL
LIN {X 0,Y 417.394,Z 388.107,A -85,B 0,C 180,E1 -10161.285,E2 -10161.285} C_VEL
LIN {X 0,Y 417.153,Z 394.043,A -85,B 0,C 180,E1 -10163.229,E2 -10163.229} C_VEL
LIN {X 0,Y 417.064,Z 398.38,A -85,B 0,C 180,E1 -10165.168,E2 -10165.168} C_VEL
LIN {X 0,Y 417.019,Z 401.252,A -85,B 0,C 180,E1 -10167.103,E2 -10167.103} C_VEL
LIN {X 0,Y 417.012,Z 402.743,A -85,B 0,C 180,E1 -10169.036,E2 -10169.036} C_VEL
LIN {X 0,Y 417.012,Z 402.89,A -85,B 0,C 180,E1 -10170.967,E2 -10170.967} C_VEL
LIN {X 0,Y 417.016,Z 401.702,A -85,B 0,C 180,E1 -10172.899,E2 -10172.899} C_VEL
LIN {X 0,Y 417.072,Z 399.165,A -85,B 0,C 180,E1 -10174.834,E2 -10174.834} C_VEL
LIN {X 0,Y 417.176,Z 395.188,A -85,B 0,C 180,E1 -10176.774,E2 -10176.774} C_VEL
LIN {X 0,Y 417.444,Z 389.654,A -85,B 0,C 180,E1 -10178.716,E2 -10178.716} C_VEL
LIN {X 0,Y 417.826,Z 383.426,A -85,B 0,C 180,E1 -10180.419,E2 -10180.419} C_VEL
LIN {X 0,Y 418.578,Z 375.683,A -85,B 0,C 180,E1 -10182.116,E2 -10182.116} C_VEL
LIN {X 0,Y 419.212,Z 367.635,A -85,B 0,C 180,E1 -10183.576,E2 -10183.576} C_VEL
LIN {X 0,Y 420.099,Z 357.959,A -85,B 0,C 180,E1 -10185.03,E2 -10185.03} C_VEL
LIN {X 0,Y 421.139,Z 347.249,A -85,B 0,C 180,E1 -10186.358,E2 -10186.358} C_VEL
LIN {X 0,Y 422.34,Z 335.416,A -85,B 0,C 180,E1 -10187.556,E2 -10187.556} C_VEL
LIN {X 0,Y 423.327,Z 323.788,A -85,B 0,C 180,E1 -10188.517,E2 -10188.517} C_VEL
LIN {X 0,Y 424.381,Z 310.251,A -85,B 0,C 180,E1 -10189.407,E2 -10189.407} C_VEL
LIN {X 0,Y 425.219,Z 297.213,A -85,B 0,C 180,E1 -10190.058,E2 -10190.058} C_VEL
LIN {X 0,Y 425.98,Z 283.206,A -85,B 0,C 180,E1 -10190.556,E2 -10190.556} C_VEL
LIN {X 0,Y 426.444,Z 268.623,A -85,B 0,C 180,E1 -10190.88,E2 -10190.88} C_VEL
LIN {X 0,Y 427.934,Z 168.623,A -85,B 0,C 180,E1 -10192.618,E2 -10192.618} C_VEL
LIN {X 0,Y 423.902,Z 147.294,A -85,B 0,C 180,E1 -10193.276,E2 -10193.276} C_VEL
LIN {X 0,Y 422.112,Z 139.199,A -85,B 0,C 180,E1 -10193.554,E2 -10193.554} C_VEL
LIN {X 0,Y 423.247,Z 125.846,A -85,B 0,C 180,E1 -10196.028,E2 -10196.028} C_VEL
LIN {X 0,Y 420.91,Z 114.549,A -85,B 0,C 180,E1 -10198.417,E2 -10198.417} C_VEL
LIN {X 0,Y 418.256,Z 104.012,A -85,B 0,C 180,E1 -10200.802,E2 -10200.802} C_VEL
LIN {X 0,Y 418.246,Z 104.018,A -85,B 0,C 180,E1 -10203.679,E2 -10203.679} C_VEL
LIN {X 0,Y 418.251,Z 104.006,A -85,B 0,C 180,E1 -10207.224,E2 -10207.224} C_VEL
LIN {X 0,Y 418.242,Z 104.01,A -85,B 0,C 180,E1 -10209.684,E2 -10209.684} C_VEL
LIN {X 0,Y 418.237,Z 104.013,A -85,B 0,C 180,E1 -10212.32,E2 -10212.32} C_VEL
LIN {X 0,Y 418.25,Z 104.009,A -85,B 0,C 180,E1 -10215.108,E2 -10215.108} C_VEL
LIN {X 0,Y 418.252,Z 104.002,A -85,B 0,C 180,E1 -10217.766,E2 -10217.766} C_VEL
LIN {X 0,Y 418.252,Z 104.014,A -85,B 0,C 180,E1 -10221.556,E2 -10221.556} C_VEL
LIN {X 0,Y 418.265,Z 104.009,A -85,B 0,C 180,E1 -10225.157,E2 -10225.157} C_VEL
LIN {X 0,Y 418.258,Z 104.012,A -85,B 0,C 180,E1 -10227.471,E2 -10227.471} C_VEL
LIN {X 0,Y 418.277,Z 104.008,A -85,B 0,C 180,E1 -10230.896,E2 -10230.896} C_VEL
LIN {X 0,Y 418.251,Z 104.009,A -85,B 0,C 180,E1 -10234.092,E2 -10234.092} C_VEL
LIN {X 0,Y 418.245,Z 104.014,A -85,B 0,C 180,E1 -10237.262,E2 -10237.262} C_VEL
LIN {X 0,Y 418.296,Z 103.997,A -85,B 0,C 180,E1 -10240.362,E2 -10240.362} C_VEL
LIN {X 0,Y 418.329,Z 103.994,A -85,B 0,C 180,E1 -10243.402,E2 -10243.402} C_VEL
LIN {X 0,Y 418.358,Z 103.994,A -85,B 0,C 180,E1 -10246.997,E2 -10246.997} C_VEL
LIN {X 0,Y 418.349,Z 104,A -85,B 0,C 180,E1 -10250.326,E2 -10250.326} C_VEL
LIN {X 0,Y 418.454,Z 103.98,A -85,B 0,C 180,E1 -10253.245,E2 -10253.245} C_VEL
LIN {X 0,Y 418.337,Z 103.997,A -85,B 0,C 180,E1 -10255.179,E2 -10255.179} C_VEL
LIN {X 0,Y 418.547,Z 103.971,A -85,B 0,C 180,E1 -10258.072,E2 -10258.072} C_VEL
LIN {X 0,Y 418.674,Z 103.958,A -85,B 0,C 180,E1 -10259.997,E2 -10259.997} C_VEL
LIN {X 0,Y 418.499,Z 103.978,A -85,B 0,C 180,E1 -10262.885,E2 -10262.885} C_VEL
LIN {X 0,Y 418.462,Z 103.98,A -85,B 0,C 180,E1 -10266.518,E2 -10266.518} C_VEL
LIN {X 0,Y 418.342,Z 103.996,A -85,B 0,C 180,E1 -10269.668,E2 -10269.668} C_VEL
LIN {X 0,Y 418.348,Z 103.994,A -85,B 0,C 180,E1 -10272.997,E2 -10272.997} C_VEL
LIN {X 0,Y 418.312,Z 103.998,A -85,B 0,C 180,E1 -10276.731,E2 -10276.731} C_VEL
LIN {X 0,Y 418.268,Z 104.004,A -85,B 0,C 180,E1 -10279.786,E2 -10279.786} C_VEL
LIN {X 0,Y 418.227,Z 104.013,A -85,B 0,C 180,E1 -10282.732,E2 -10282.732} C_VEL
LIN {X 0,Y 418.254,Z 104.005,A -85,B 0,C 180,E1 -10285.901,E2 -10285.901} C_VEL
LIN {X 0,Y 418.261,Z 103.999,A -85,B 0,C 180,E1 -10289.1,E2 -10289.1} C_VEL
LIN {X 0,Y 418.246,Z 104.01,A -85,B 0,C 180,E1 -10292.84,E2 -10292.84} C_VEL
LIN {X 0,Y 418.231,Z 104.015,A -85,B 0,C 180,E1 -10296.233,E2 -10296.233} C_VEL
LIN {X 0,Y 418.23,Z 104.014,A -85,B 0,C 180,E1 -10299.679,E2 -10299.679} C_VEL
LIN {X 0,Y 418.213,Z 104.019,A -85,B 0,C 180,E1 -10302.317,E2 -10302.317} C_VEL
LIN {X 0,Y 418.217,Z 104.014,A -85,B 0,C 180,E1 -10305.105,E2 -10305.105} C_VEL
LIN {X 0,Y 418.251,Z 104.212,A -85,B 0,C 180,E1 -10306.845,E2 -10306.845} C_VEL
LIN {X 0,Y 420.906,Z 115.571,A -85,B 0,C 180,E1 -10309.625,E2 -10309.625} C_VEL
LIN {X 0,Y 421.63,Z 119.138,A -85,B 0,C 180,E1 -10310.463,E2 -10310.463} C_VEL
LIN {X 0,Y 424.675,Z 127.065,A -85,B 0,C 180,E1 -10310.823,E2 -10310.823} C_VEL
LIN {X 0,Y 428.417,Z 143.235,A -85,B 0,C 180,E1 -10311.371,E2 -10311.371} C_VEL
LIN {X 0,Y 426.463,Z 256.177,A -85,B 0,C 180,E1 -10313.352,E2 -10313.352} C_VEL
LIN {X 0,Y 425.925,Z 270.308,A -85,B 0,C 180,E1 -10313.791,E2 -10313.791} C_VEL
LIN {X 0,Y 425.26,Z 283.226,A -85,B 0,C 180,E1 -10314.37,E2 -10314.37} C_VEL
LIN {X 0,Y 424.357,Z 296.398,A -85,B 0,C 180,E1 -10315.153,E2 -10315.153} C_VEL
LIN {X 0,Y 423.399,Z 308.684,A -85,B 0,C 180,E1 -10316.085,E2 -10316.085} C_VEL
LIN {X 0,Y 422.271,Z 321.061,A -85,B 0,C 180,E1 -10317.253,E2 -10317.253} C_VEL
LIN {X 0,Y 421.24,Z 331.749,A -85,B 0,C 180,E1 -10318.492,E2 -10318.492} C_VEL
LIN {X 0,Y 420.26,Z 341.691,A -85,B 0,C 180,E1 -10319.887,E2 -10319.887} C_VEL
LIN {X 0,Y 419.299,Z 350.951,A -85,B 0,C 180,E1 -10321.464,E2 -10321.464} C_VEL
LIN {X 0,Y 418.586,Z 358.513,A -85,B 0,C 180,E1 -10323.041,E2 -10323.041} C_VEL
LIN {X 0,Y 418.014,Z 364.664,A -85,B 0,C 180,E1 -10324.612,E2 -10324.612} C_VEL
LIN {X 0,Y 417.615,Z 369.621,A -85,B 0,C 180,E1 -10326.177,E2 -10326.177} C_VEL
LIN {X 0,Y 417.377,Z 373.716,A -85,B 0,C 180,E1 -10327.824,E2 -10327.824} C_VEL
LIN {X 0,Y 417.143,Z 376.476,A -85,B 0,C 180,E1 -10329.278,E2 -10329.278} C_VEL
LIN {X 0,Y 416.936,Z 378.977,A -85,B 0,C 180,E1 -10331.319,E2 -10331.319} C_VEL
LIN {X 0,Y 416.895,Z 380.004,A -85,B 0,C 180,E1 -10333.345,E2 -10333.345} C_VEL
LIN {X 0,Y 416.875,Z 379.609,A -85,B 0,C 180,E1 -10335.351,E2 -10335.351} C_VEL
LIN {X 0,Y 416.956,Z 377.814,A -85,B 0,C 180,E1 -10337.341,E2 -10337.341} C_VEL
LIN {X 0,Y 416.985,Z 377.443,A -85,B 0,C 180,E1 -10337.613,E2 -10337.613} C_VEL
LIN {X 0,Y 416.41,Z 376.299,A -85,B 0,C 180,E1 -10338.405,E2 -10338.405} C_VEL
LIN {X 0,Y 413.676,Z 373.992,A -85,B 0,C 180,E1 -10339.683,E2 -10339.683} C_VEL
LIN {X 0,Y 411.365,Z 371.749,A -85,B 0,C 180,E1 -10340.698,E2 -10340.698} C_VEL
LIN {X 0,Y 410.427,Z 369.768,A -85,B 0,C 180,E1 -10341.468,E2 -10341.468} C_VEL
LIN {X 0,Y 410.382,Z 369.019,A -85,B 0,C 180,E1 -10341.725,E2 -10341.725} C_VEL
LIN {X 0,Y 410.848,Z 362.707,A -85,B 0,C 180,E1 -10343.615,E2 -10343.615} C_VEL
LIN {X 0,Y 411.348,Z 355.4,A -85,B 0,C 180,E1 -10345.344,E2 -10345.344} C_VEL
LIN {X 0,Y 412.13,Z 346.324,A -85,B 0,C 180,E1 -10347.066,E2 -10347.066} C_VEL
LIN {X 0,Y 412.958,Z 336.834,A -85,B 0,C 180,E1 -10348.536,E2 -10348.536} C_VEL
LIN {X 0,Y 413.849,Z 326.346,A -85,B 0,C 180,E1 -10349.877,E2 -10349.877} C_VEL
LIN {X 0,Y 414.764,Z 314.879,A -85,B 0,C 180,E1 -10351.082,E2 -10351.082} C_VEL
LIN {X 0,Y 415.748,Z 301.939,A -85,B 0,C 180,E1 -10352.178,E2 -10352.178} C_VEL
LIN {X 0,Y 416.616,Z 288.41,A -85,B 0,C 180,E1 -10353.081,E2 -10353.081} C_VEL
LIN {X 0,Y 417.233,Z 275.449,A -85,B 0,C 180,E1 -10353.741,E2 -10353.741} C_VEL
